// TwinCAT 3 PLC project CNM_ProductionMetrics
// Title: CNM_ProductionMetrics
// Company: ekvip automation GmbH
// Author: tsch
// ProjectVersion: 0.1.1.0
// Description: This library contains classes for measuring and storing production statistics like part counter and cycle time recorder.
// ProgramVersion: 3.1.4026.19
// libraries:
//   CNM_AbstractObject, * (ekvip automation GmbH)
//   CNM_Collections, * (ekvip automation GmbH)
//   CNM_CommandInterfaces, * (ekvip automation GmbH)
//   CNM_ConcreteMessages, * (ekvip automation GmbH)
//   CNM_CycleManager, * (ekvip automation GmbH)
//   CNM_OpModeHandling, * (ekvip automation GmbH)
//   CNM_ProductionMetricInterfaces, * (ekvip automation GmbH)
//   CNM_ReturnTypes, * (ekvip automation GmbH)
//   Tc2_System, * (Beckhoff Automation GmbH)
// project tree:
//   classes/Data/ CycleTimeData.TcPOU, MeasurementData.TcPOU, PartTrackingData.TcPOU
//   classes/Measurements/CycleTimeRecorder/commands/ CycleTimeCaptureCycleCommand.TcPOU, CycleTimeRecorderCommands.TcPOU, CycleTimeStartCycleCommand.TcPOU
//   classes/Measurements/CycleTimeRecorder/ CycleTimeRecorder.TcPOU, CycleTimeRecorderConfiguration.TcPOU
//   classes/Measurements/PartTracking/Commands/ PartTrackingCommands.TcPOU, PartTrackingProcssingStartedCommand.TcPOU, PartTrackingProcssingDoneCommand.TcPOU
//   classes/Measurements/PartTracking/ PartTrackingConfiguration.TcPOU, PartTrackingRecorder.TcPOU
//   classes/Measurements/SimpleMeasurement/commands/ MeasurementAddEntryCommand.TcPOU, MeasurementRecorderCommands.TcPOU
//   classes/Measurements/SimpleMeasurement/ DefaultMeasurementConfiguration.TcPOU, MeasurementRecorder.TcPOU
//   Functions/ GetCurrentLTimeStamp.TcPOU
//   Project Information/ F_GetCompany.TcPOU, F_GetTitle.TcPOU, F_GetVersion.TcPOU
//   / Settings.TcGVL
//   Version/ Global_Version.TcGVL

// ---- Settings.TcGVL
{attribute 'qualified_only'}
VAR_GLOBAL CONSTANT
	(*
	 	The size of the internal queue in the data recorders. 
		when the queue is full, an alarm will be raised and no other 
		dataset will be queued until the list gets emptied 
	*)
	QUEUE_SIZE_FOR_DATA_RECORDS_PER_RECORDER :UDINT := 3;
END_VAR

// ---- Version/Global_Version.TcGVL
{attribute 'TcGenerated'}
{attribute 'no-analysis'}
{attribute 'linkalways'}
// This function has been automatically generated from the project information.
VAR_GLOBAL CONSTANT
	{attribute 'const_non_replaced'}
	stLibVersion_CNM_ProductionMetrics : ST_LibVersion := (iMajor := 0, iMinor := 1, iBuild := 1, iRevision := 0, nFlags := 0, sVersion := '0.1.1.0');
END_VAR

// ---- classes/Data/CycleTimeData.TcPOU
(*

## Short summary

This class serves as a pure data transfer object and can be used to create a new cycle time data set.
An instance of this class can be appended to a production data set list.

.. <legal notes>

legal notes
=================
| SPDX-FileCopyrightText: © 2022 ekvip automation GmbH <info@ekvip.de>
| SPDX-License-Identifier: Apache-2.0
| For details check: Apache-2.0_

.. _Apache-2.0: https://www.apache.org/licenses/LICENSE-2.0

.. </legal notes>

*)
{attribute 'enable_dynamic_creation'}
FUNCTION_BLOCK CycleTimeData EXTENDS CNM_AbstractObject.Object IMPLEMENTS CNM_ProductionMetricInterfaces.ICycleTimeData
VAR
	data :CNM_ProductionMetricInterfaces.CycleTimeDataStruct;
END_VAR

(*

## Short summary

This abstract property returns the class name of the concrete object, 
which is useful for logging/debugging purpose or to check the class name
for ``__DELETE`` in factories (sometimes it's necessary to do more 
than just to free the memory).

.. <legal notes>

legal notes
=================
| SPDX-FileCopyrightText: © 2022 ekvip automation GmbH <info@ekvip.de>
| SPDX-License-Identifier: Apache-2.0
| For details check: Apache-2.0_

.. _Apache-2.0: https://www.apache.org/licenses/LICENSE-2.0

.. </legal notes>

*)
PROPERTY className : CNM_AbstractObject.ClassName
GET
className := 'CycleTimeData';
END_GET
END_PROPERTY

PROPERTY dataset : CNM_ProductionMetricInterfaces.CycleTimeDataStruct
GET
dataset := THIS^.data;
END_GET
END_PROPERTY

(*

## Short summary

The constructor ``FB_init`` is needed to create an unique hash code.
The hash code is a pseudo random number create with a [xorshift](https://en.wikipedia.org/wiki/Xorshift) algorithm.
It can be overwritten on derivations, because it will be called implicit, ``SUPER^.FB_init()`` is not required.
For more information check: [Behavoir with derived function blocks](https://infosys.beckhoff.com/content/1033/tc3_plc_intro/5482088715.html?id=6983869892358031022)

.. <legal notes>

legal notes
=================
| SPDX-FileCopyrightText: © 2022 ekvip automation GmbH <info@ekvip.de>
| SPDX-License-Identifier: Apache-2.0
| For details check: Apache-2.0_

.. _Apache-2.0: https://www.apache.org/licenses/LICENSE-2.0

.. </legal notes>



*)
METHOD FB_init : BOOL
VAR_INPUT
	(* if TRUE, the retain variables are initialized (warm start / cold start)*)
	bInitRetains	: BOOL;
	(* if TRUE, the instance afterwards gets moved into the copy code (online change) *)
	bInCopyCode	: BOOL;
	(* the data set this instance should capsulate *)
	data :CNM_ProductionMetricInterfaces.CycleTimeDataStruct;
END_VAR
THIS^.data := data;
END_METHOD

END_FUNCTION_BLOCK

// ---- classes/Data/MeasurementData.TcPOU
(*
## Short summary

This class serves as a pure data transfer object and can be used to create a new measurement data set.
An instance of this class can be appended to a production data set list.

.. <legal notes>

legal notes
=================
| SPDX-FileCopyrightText: © 2022 ekvip automation GmbH <info@ekvip.de>
| SPDX-License-Identifier: Apache-2.0
| For details check: Apache-2.0_

.. _Apache-2.0: https://www.apache.org/licenses/LICENSE-2.0

.. </legal notes>

*)
{attribute 'enable_dynamic_creation'}
FUNCTION_BLOCK MeasurementData EXTENDS CNM_AbstractObject.Object IMPLEMENTS CNM_ProductionMetricInterfaces.IMeasurementData
VAR
	data : CNM_ProductionMetricInterfaces.MeasurementEntryStruct;
END_VAR

(*

## Short summary

This abstract property returns the class name of the concrete object, 
which is useful for logging/debugging purpose or to check the class name
for ``__DELETE`` in factories (sometimes it's necessary to do more 
than just to free the memory).

.. <legal notes>

legal notes
=================
| SPDX-FileCopyrightText: © 2022 ekvip automation GmbH <info@ekvip.de>
| SPDX-License-Identifier: Apache-2.0
| For details check: Apache-2.0_

.. _Apache-2.0: https://www.apache.org/licenses/LICENSE-2.0

.. </legal notes>

*)
PROPERTY className : CNM_AbstractObject.ClassName
GET
className := 'MeasurementData';
END_GET
END_PROPERTY

(*
## Short summary

This property returns a measurement data set.

.. <legal notes>

legal notes
=================
| SPDX-FileCopyrightText: © 2025 ekvip automation GmbH <info@ekvip.de>
| SPDX-License-Identifier: Apache-2.0
| For details check: Apache-2.0_

.. _Apache-2.0: https://www.apache.org/licenses/LICENSE-2.0

.. </legal notes>

*)
PROPERTY dataset : CNM_ProductionMetricInterfaces.MeasurementEntryStruct
GET
dataset := THIS^.data;
END_GET
END_PROPERTY

(*

## Short summary

The constructor ``FB_init`` is needed to create an unique hash code.
The hash code is a pseudo random number create with a [xorshift](https://en.wikipedia.org/wiki/Xorshift) algorithm.
It can be overwritten on derivations, because it will be called implicit, ``SUPER^.FB_init()`` is not required.
For more information check: [Behavoir with derived function blocks](https://infosys.beckhoff.com/content/1033/tc3_plc_intro/5482088715.html?id=6983869892358031022)

.. <legal notes>

legal notes
=================
| SPDX-FileCopyrightText: © 2022 ekvip automation GmbH <info@ekvip.de>
| SPDX-License-Identifier: Apache-2.0
| For details check: Apache-2.0_

.. _Apache-2.0: https://www.apache.org/licenses/LICENSE-2.0

.. </legal notes>



*)
METHOD FB_init : BOOL
VAR_INPUT
	(* if TRUE, the retain variables are initialized (warm start / cold start)*)
	bInitRetains	: BOOL;
	(* if TRUE, the instance afterwards gets moved into the copy code (online change) *)
	bInCopyCode	: BOOL;
	(* the data set this instance should capsulate *)
	data :CNM_ProductionMetricInterfaces.MeasurementEntryStruct;
END_VAR
THIS^.data := data;
END_METHOD

END_FUNCTION_BLOCK

// ---- classes/Data/PartTrackingData.TcPOU
(*

## Short summary

This class serves as a pure data transfer object and can be used to create a new part counter data set.
An instance of this class can be appended to a production data set list.

.. <legal notes>

legal notes
=================
| SPDX-FileCopyrightText: © 2022 ekvip automation GmbH <info@ekvip.de>
| SPDX-License-Identifier: Apache-2.0
| For details check: Apache-2.0_

.. _Apache-2.0: https://www.apache.org/licenses/LICENSE-2.0

.. </legal notes>

*)
{attribute 'enable_dynamic_creation'}
FUNCTION_BLOCK PartTrackingData EXTENDS CNM_AbstractObject.Object IMPLEMENTS CNM_ProductionMetricInterfaces.IPartTrackingData
VAR
	data :CNM_ProductionMetricInterfaces.PartDataTrackingStruct;
END_VAR

(*

## Short summary

This abstract property returns the class name of the concrete object, 
which is useful for logging/debugging purpose or to check the class name
for ``__DELETE`` in factories (sometimes it's necessary to do more 
than just to free the memory).

.. <legal notes>

legal notes
=================
| SPDX-FileCopyrightText: © 2022 ekvip automation GmbH <info@ekvip.de>
| SPDX-License-Identifier: Apache-2.0
| For details check: Apache-2.0_

.. _Apache-2.0: https://www.apache.org/licenses/LICENSE-2.0

.. </legal notes>

*)
PROPERTY className : CNM_AbstractObject.ClassName
GET
className := 'PartCounterData';
END_GET
END_PROPERTY

PROPERTY dataset : CNM_ProductionMetricInterfaces.PartDataTrackingStruct
GET
dataset := THIS^.data;
END_GET
END_PROPERTY

(*

## Short summary

The constructor ``FB_init`` is needed to create an unique hash code.
The hash code is a pseudo random number create with a [xorshift](https://en.wikipedia.org/wiki/Xorshift) algorithm.
It can be overwritten on derivations, because it will be called implicit, ``SUPER^.FB_init()`` is not required.
For more information check: [Behavoir with derived function blocks](https://infosys.beckhoff.com/content/1033/tc3_plc_intro/5482088715.html?id=6983869892358031022)

.. <legal notes>

legal notes
=================
| SPDX-FileCopyrightText: © 2022 ekvip automation GmbH <info@ekvip.de>
| SPDX-License-Identifier: Apache-2.0
| For details check: Apache-2.0_

.. _Apache-2.0: https://www.apache.org/licenses/LICENSE-2.0

.. </legal notes>



*)
METHOD FB_init : BOOL
VAR_INPUT
	(* if TRUE, the retain variables are initialized (warm start / cold start)*)
	bInitRetains	: BOOL;
	(* if TRUE, the instance afterwards gets moved into the copy code (online change) *)
	bInCopyCode	: BOOL;
	(* the data set this instance should capsulate *)
	data :CNM_ProductionMetricInterfaces.PartDataTrackingStruct;
END_VAR
THIS^.data := data;
END_METHOD

END_FUNCTION_BLOCK

// ---- classes/Measurements/CycleTimeRecorder/commands/CycleTimeCaptureCycleCommand.TcPOU
(*
## Short summary

This command can be used to set the cycle start timestamp manually.

**Attention:** If only the captureCurrentCycle method is called, the start timestamp will be set automatically when the previous cycle is done.

.. <legal notes>

legal notes
=================
| SPDX-FileCopyrightText: © 2025 ekvip automation GmbH <info@ekvip.de>
| SPDX-License-Identifier: Apache-2.0
| For details check: Apache-2.0_

.. _Apache-2.0: https://www.apache.org/licenses/LICENSE-2.0

.. </legal notes>

*)
FUNCTION_BLOCK CycleTimeCaptureCycleCommand EXTENDS CNM_AbstractObject.Object IMPLEMENTS CNM_CommandInterfaces.ISingleAttempt
VAR
	recorder :CNM_ProductionMetricInterfaces.ICycleTimeRecorder;
	additionalMessage :Tc2_System.T_MaxString := '';
END_VAR

(*

## Short summary

This abstract property returns the class name of the concrete object, 
which is useful for logging/debugging purpose or to check the class name
for ``__DELETE`` in factories (sometimes it's necessary to do more 
than just to free the memory).

.. <legal notes>

legal notes
=================
| SPDX-FileCopyrightText: © 2022 ekvip automation GmbH <info@ekvip.de>
| SPDX-License-Identifier: Apache-2.0
| For details check: Apache-2.0_

.. _Apache-2.0: https://www.apache.org/licenses/LICENSE-2.0

.. </legal notes>

*)
PROPERTY className : CNM_AbstractObject.ClassName
GET
className :=  'CNM_ProductionMetrics.CycleTimeCaptureCycleCommand';
END_GET
END_PROPERTY

(*

## Short summary

Invokes the action associated with this interface.

.. <legal notes>

legal notes
=================
| SPDX-FileCopyrightText: © 2024 ekvip automation GmbH <info@ekvip.de>
| SPDX-License-Identifier: Apache-2.0
| For details check: Apache-2.0_

.. _Apache-2.0: https://www.apache.org/licenses/LICENSE-2.0

.. </legal notes>



*)
METHOD invoke : CNM_ReturnTypes.SingleExecutionResult
IF THIS^.isObjectValid(THIS^.recorder) THEN
	invoke := THIS^.recorder.captureCurrentCycle(additionalMessage := THIS^.additionalMessage);
ELSE
	invoke := CNM_ReturnTypes.SingleExecutionResult.ABORTED;
END_IF
END_METHOD

METHOD INTERNAL setParameters
VAR_INPUT
	(* can be used to provide additional informations for the record, e.g. multiple measurements neccesray or test part *)
	additionalMessage	:Tc2_System.T_MaxString := '';
END_VAR
THIS^.additionalMessage := additionalMessage;
END_METHOD

(*
## Short summary

This methods sets the cycletime recorder interface on which the command is executed.

.. <legal notes>

legal notes
=================
| SPDX-FileCopyrightText: © 2025 ekvip automation GmbH <info@ekvip.de>
| SPDX-License-Identifier: Apache-2.0
| For details check: Apache-2.0_

.. _Apache-2.0: https://www.apache.org/licenses/LICENSE-2.0

.. </legal notes>

*)

METHOD INTERNAL setRecorder
VAR_INPUT
	recorder :CNM_ProductionMetricInterfaces.ICycleTimeRecorder;
END_VAR
IF THIS^.isObjectValid(recorder) THEN
	THIS^.recorder := recorder;
END_IF
END_METHOD

END_FUNCTION_BLOCK

// ---- classes/Measurements/CycleTimeRecorder/commands/CycleTimeRecorderCommands.TcPOU
(* 
## Short summary

This class is a collection of cycle time recorder commands that provides a fluent interface for single attempt commands, which can be evaluated by a cycle manager instance.
### Example 
```
	cycleManager.leave(
		cycleTimeRecorder.commands.captureCurrentCycle(
			additionalMessage := 'just an example'
		)
	);  
	```

.. <legal notes>

legal notes
=================
| SPDX-FileCopyrightText: © 2025 ekvip automation GmbH <info@ekvip.de>
| SPDX-License-Identifier: Apache-2.0
| For details check: Apache-2.0_

.. _Apache-2.0: https://www.apache.org/licenses/LICENSE-2.0

.. </legal notes>
	
*)

FUNCTION_BLOCK CycleTimeRecorderCommands EXTENDS CNM_AbstractObject.Object IMPLEMENTS CNM_ProductionMetricInterfaces.ICycleTimeRecorderCommands
VAR
	captureCommand :CycleTimeCaptureCycleCommand;
	startCycleCommand :CycleTimeStartCycleCommand;
END_VAR

(*

## Short summary

This command creates a new cycle time roecord for the currently produced part by calculating the the passed time since the last call of this method.
If a new mode is started the last timestamp will be set to the moment when the mode was started.


.. <legal notes>

legal notes
=================
| SPDX-FileCopyrightText: © 2025 ekvip automation GmbH <info@ekvip.de>
| SPDX-License-Identifier: Apache-2.0
| For details check: Apache-2.0_

.. _Apache-2.0: https://www.apache.org/licenses/LICENSE-2.0

.. </legal notes>

*)
METHOD captureCurrentCycle : CNM_CommandInterfaces.ISingleAttempt
VAR_INPUT
	(* can be used to provide additional informations for the record, e.g. multiple measurements neccesray or test part *)
	additionalMessage	: Tc2_System.T_MaxString := '';
END_VAR
THIS^.captureCommand.setParameters(additionalMessage);
captureCurrentCycle := THIS^.captureCommand;
END_METHOD

(*

## Short summary

This abstract property returns the class name of the concrete object, 
which is useful for logging/debugging purpose or to check the class name
for ``__DELETE`` in factories (sometimes it's necessary to do more 
than just to free the memory).

.. <legal notes>

legal notes
=================
| SPDX-FileCopyrightText: © 2022 ekvip automation GmbH <info@ekvip.de>
| SPDX-License-Identifier: Apache-2.0
| For details check: Apache-2.0_

.. _Apache-2.0: https://www.apache.org/licenses/LICENSE-2.0

.. </legal notes>

*)

PROPERTY className : CNM_AbstractObject.ClassName
GET
 className := 'CNM_ProductionMetrics.CycleTimeRecorderCommands';
END_GET
END_PROPERTY

METHOD INTERNAL setRecorder : BOOL
VAR_INPUT
	recorder :CNM_ProductionMetricInterfaces.ICycleTimeRecorder;
END_VAR
IF THIS^.isObjectValid(recorder) THEN
	THIS^.captureCommand.setRecorder(recorder);
	THIS^.startCycleCommand.setRecorder(recorder);
END_IF
END_METHOD

(*
## Short summary

This command can be used to set the cycle start timestamp manually.

**Attention:** If only the captureCurrentCycle method is called, the start timestamp will be set automatically when the previous cycle is done.

.. <legal notes>

legal notes
=================
| SPDX-FileCopyrightText: © 2025 ekvip automation GmbH <info@ekvip.de>
| SPDX-License-Identifier: Apache-2.0
| For details check: Apache-2.0_

.. _Apache-2.0: https://www.apache.org/licenses/LICENSE-2.0

.. </legal notes>

*)
METHOD startCycle : CNM_CommandInterfaces.ISingleAttempt
startCycle := THIS^.startCycleCommand;
END_METHOD

END_FUNCTION_BLOCK

// ---- classes/Measurements/CycleTimeRecorder/commands/CycleTimeStartCycleCommand.TcPOU
(*
## Short summary

This command can be used to set the cycle start timestamp manually.

**Attention:** If only the captureCurrentCycle method is called, the start timestamp will be set automatically when the previous cycle is done.

.. <legal notes>

legal notes
=================
| SPDX-FileCopyrightText: © 2025 ekvip automation GmbH <info@ekvip.de>
| SPDX-License-Identifier: Apache-2.0
| For details check: Apache-2.0_

.. _Apache-2.0: https://www.apache.org/licenses/LICENSE-2.0

.. </legal notes>

*)
FUNCTION_BLOCK CycleTimeStartCycleCommand EXTENDS CNM_AbstractObject.Object IMPLEMENTS CNM_CommandInterfaces.ISingleAttempt
VAR
	recorder :CNM_ProductionMetricInterfaces.ICycleTimeRecorder;
END_VAR

(*

## Short summary

This abstract property returns the class name of the concrete object, 
which is useful for logging/debugging purpose or to check the class name
for ``__DELETE`` in factories (sometimes it's necessary to do more 
than just to free the memory).

.. <legal notes>

legal notes
=================
| SPDX-FileCopyrightText: © 2022 ekvip automation GmbH <info@ekvip.de>
| SPDX-License-Identifier: Apache-2.0
| For details check: Apache-2.0_

.. _Apache-2.0: https://www.apache.org/licenses/LICENSE-2.0

.. </legal notes>

*)
PROPERTY className : CNM_AbstractObject.ClassName
GET
className := 'CNM_ProductionMetrics.CycleTimeStartCycleCommand';
END_GET
END_PROPERTY

(*

## Short summary

Invokes the action associated with this interface.

.. <legal notes>

legal notes
=================
| SPDX-FileCopyrightText: © 2024 ekvip automation GmbH <info@ekvip.de>
| SPDX-License-Identifier: Apache-2.0
| For details check: Apache-2.0_

.. _Apache-2.0: https://www.apache.org/licenses/LICENSE-2.0

.. </legal notes>



*)
METHOD invoke : CNM_ReturnTypes.SingleExecutionResult
IF THIS^.isObjectValid(THIS^.recorder) THEN
	invoke := THIS^.recorder.startCycle();
ELSE
	invoke := CNM_ReturnTypes.SingleExecutionResult.ABORTED;
END_IF
END_METHOD

(*
## Short summary

This methods sets the cycletime recorder interface on which the command is executed.

.. <legal notes>

legal notes
=================
| SPDX-FileCopyrightText: © 2025 ekvip automation GmbH <info@ekvip.de>
| SPDX-License-Identifier: Apache-2.0
| For details check: Apache-2.0_

.. _Apache-2.0: https://www.apache.org/licenses/LICENSE-2.0

.. </legal notes>

*)

METHOD setRecorder
VAR_INPUT
	recorder :CNM_ProductionMetricInterfaces.ICycleTimeRecorder;
END_VAR
IF THIS^.isObjectValid(recorder) THEN
	THIS^.recorder := recorder;
END_IF
END_METHOD

END_FUNCTION_BLOCK

// ---- classes/Measurements/CycleTimeRecorder/CycleTimeRecorder.TcPOU
(*
## Short summary

This class provides the functionalities to measure timespans for processes and commands.
It can measure processing times (start time -> stop time) and cycle times (last stop time -> stop time).

.. <legal notes>

legal notes
=================
| SPDX-FileCopyrightText: © 2025 ekvip automation GmbH <info@ekvip.de>
| SPDX-License-Identifier: Apache-2.0
| For details check: Apache-2.0_

.. _Apache-2.0: https://www.apache.org/licenses/LICENSE-2.0

.. </legal notes>

*)

FUNCTION_BLOCK CycleTimeRecorder EXTENDS CNM_OpModeHandler.AbstractCyclicNode IMPLEMENTS CNM_ProductionMetricInterfaces.ICycleTimeRecorder
VAR
	(* current data *)
	currentCycleTimeData :CNM_ProductionMetricInterfaces.CycleTimeDataStruct;
	(* queue for the measurements *)
	dataSetList :CNM_Collections.LinkedList;
	(* the variable that is used as data slot to provide data for the database *)
	{ attribute 'TcHmiSymbol.ShowRecursively' }
	cycleTimeRecord :CNM_ProductionMetricInterfaces.CycleTimeDataStruct;
	(* mailbox flag for the database that we have a new entry, should be reset by the server when data was read *)
	{ attribute 'TcHmiSymbol.Show' }
	newDataAvailable :BOOL := FALSE;
	(* command delegates *)
	cycleTimeCommands :CycleTimeRecorderCommands;
	(* error for failed queryInterface *)
	interfaceQueryFailedAlarm :CNM_ConcreteMessages.TcError(
		event := Global.TC_EVENTS.MemoryErrors.CycleTimeRecorderQueryInterfacFailed , 
		injectedService := THIS^.messageService
	); 
	(* error for maximum queue size *)
	maxQueueSizeAlarm :CNM_ConcreteMessages.TcError(event := Global.TC_EVENTS.MemoryErrors.CycleTimeMaxQueueSize, injectedService := THIS^.messageService);
END_VAR

(*

## Short summary

This method creates a new cycle time roecord for the currently produced part by calculating the the passed time since the last call of this method.
If a new mode is started the last timestamp will be set to the moment when the mode was started.


.. <legal notes>

legal notes
=================
| SPDX-FileCopyrightText: © 2025 ekvip automation GmbH <info@ekvip.de>
| SPDX-License-Identifier: Apache-2.0
| For details check: Apache-2.0_

.. _Apache-2.0: https://www.apache.org/licenses/LICENSE-2.0

.. </legal notes>

*)
METHOD captureCurrentCycle : CNM_ProductionMetricInterfaces.CNM_ReturnTypes.SingleExecutionResult
VAR_INPUT
	(* can be used to provide additional informations for the record, e.g. multiple measurements neccesray or test part *)
	additionalMessage	: Tc2_System.T_MaxString := '';
END_VAR
VAR
	dto :POINTER TO CycleTimeData;
	(* data backup to restore timestamps *)
	backupEndTimestamp :LDT;
END_VAR
captureCurrentCycle := CNM_ReturnTypes.SingleExecutionResult.ABORTED;
// check if we can queue the dataset - throw error if the max queuesize is reached
IF ( THIS^.dataSetList.size >= THIS^.maxQueueSize ) THEN
	THIS^.maxQueueSizeAlarm.throw();
	RETURN;
END_IF

backupEndTimestamp  := THIS^.currentCycleTimeData.endTimestamp;
THIS^.currentCycleTimeData.cycleTime := 
	SEL(
		TO_UDINT(THIS^.currentCycleTimeData.endTimestamp) > 0, 
		TO_LTIME(0), 
		TO_LTIME(GetCurrentLTimeStamp() - THIS^.currentCycleTimeData.endTimestamp ));
THIS^.currentCycleTimeData.endTimestamp := GetCurrentLTimeStamp();
THIS^.currentCycleTimeData.processingTime := 
	SEL(
		TO_UDINT(THIS^.currentCycleTimeData.startTimestamp) > 0, 
		TO_LTIME(0), 
		TO_LTIME(THIS^.currentCycleTimeData.endTimestamp - THIS^.currentCycleTimeData.startTimestamp));
THIS^.currentCycleTimeData.process := THIS^.configuration.process;
THIS^.currentCycleTimeData.productType := THIS^.configuration.productType;
THIS^.currentCycleTimeData.targetCycletime := THIS^.configuration.targetCycleTime;
THIS^.currentCycleTimeData.additionalMessage := additionalMessage;
dto := __NEW(CycleTimeData(data := THIS^.currentCycleTimeData));
IF (dto <> 0) THEN
	captureCurrentCycle := THIS^.dataSetList.append(dto^);
ELSE
	// restore data for retry
	THIS^.currentCycleTimeData.endTimestamp := backupEndTimestamp;
END_IF
END_METHOD

(*

## Short summary

This abstract property returns the class name of the concrete object, 
which is useful for logging/debugging purpose or to check the class name
for ``__DELETE`` in factories (sometimes it's necessary to do more 
than just to free the memory).

.. <legal notes>

legal notes
=================
| SPDX-FileCopyrightText: © 2022 ekvip automation GmbH <info@ekvip.de>
| SPDX-License-Identifier: Apache-2.0
| For details check: Apache-2.0_

.. _Apache-2.0: https://www.apache.org/licenses/LICENSE-2.0

.. </legal notes>

*)
PROPERTY className : CNM_AbstractObject.ClassName
GET
className := 'CycleTimeRecorder';
END_GET
END_PROPERTY

(* 
## Short summary

This is a fluent interface that provides single attempt commands, which can be evaluated by a cycle manager instance.
### Example 
```
	cycleManager.leave(
		cycleTimeRecorder.commands.captureCurrentCycle(
			additionalMessage := 'just an example'
		)
	);  
	```

.. <legal notes>

legal notes
=================
| SPDX-FileCopyrightText: © 2025 ekvip automation GmbH <info@ekvip.de>
| SPDX-License-Identifier: Apache-2.0
| For details check: Apache-2.0_

.. _Apache-2.0: https://www.apache.org/licenses/LICENSE-2.0

.. </legal notes>
	
*)

PROPERTY commands : CNM_ProductionMetricInterfaces.ICycleTimeRecorderCommands
GET
commands := THIS^.cycleTimeCommands;
END_GET
END_PROPERTY

(*
## Short summary

This property returns an fluent interface for the cycle time recorder configuration.
The following things should be configured after a type / product / batch change was performed:
 -product type: either the name of the overall product or the individual feed parts to be processed
 -targetCycleTime: the target cycle time for this process and product type
 
The process name can be set once during the initialization of the PLC as it usually doesn't change.

.. <legal notes>

legal notes
=================
| SPDX-FileCopyrightText: © 2025 ekvip automation GmbH <info@ekvip.de>
| SPDX-License-Identifier: Apache-2.0
| For details check: Apache-2.0_

.. _Apache-2.0: https://www.apache.org/licenses/LICENSE-2.0

.. </legal notes>

*)
PROPERTY configuration : CNM_ProductionMetricInterfaces.ICycleTimeConfiguration
GET
VAR_INST
	config :CycleTimeRecorderConfiguration;
END_VAR
configuration := config;
END_GET
END_PROPERTY

(* 
## Short summary

This method disables a node (E.g. axes should be disabled). It can take mutliple cycles. It has to be implemented for every node/device.
The execute input needs a rising edge to execute the method.
If there is nothing to disable, just return a 'SUCCESS' state.

This method is called automatically by the operation mode handler.

.. <legal notes>

legal notes
=================
| SPDX-FileCopyrightText: © 2024 ekvip automation GmbH <info@ekvip.de>
| SPDX-License-Identifier: Apache-2.0
| For details check: Apache-2.0_

.. _Apache-2.0: https://www.apache.org/licenses/LICENSE-2.0

.. </legal notes>

*)
METHOD disable : CNM_ReturnTypes.SingleExecutionState
VAR_INPUT
	execute	: BOOL;
END_VAR
// nothing to disable
disable := CNM_ReturnTypes.SingleExecutionState.SUCCESS;
END_METHOD

(* 
## Short summary

This method enables a node. It can take mutliple cycles. It has to be implemented for every node/device.
The intention is to enable devices here, e.g. axes, laser, dispenser etc.
The execute input needs a rising edge to execute the method.
If there is nothing to enable, just return a 'SUCCESS' state.

This method is called automatically by the operation mode handler.

.. <legal notes>

legal notes
=================
| SPDX-FileCopyrightText: © 2024 ekvip automation GmbH <info@ekvip.de>
| SPDX-License-Identifier: Apache-2.0
| For details check: Apache-2.0_

.. _Apache-2.0: https://www.apache.org/licenses/LICENSE-2.0

.. </legal notes>

*)
METHOD enable : CNM_ReturnTypes.SingleExecutionState
VAR_INPUT
	execute	: BOOL;
END_VAR
// nothing to enable
enable := CNM_ReturnTypes.SingleExecutionState.SUCCESS;
END_METHOD

(*

## Short summary

The constructor ``FB_init`` is needed to create an unique hash code.
The hash code is a pseudo random number create with a [xorshift](https://en.wikipedia.org/wiki/Xorshift) algorithm.
It can be overwritten on derivations, because it will be called implicit, ``SUPER^.FB_init()`` is not required.
For more information check: [Behavoir with derived function blocks](https://infosys.beckhoff.com/content/1033/tc3_plc_intro/5482088715.html?id=6983869892358031022)

.. <legal notes>

legal notes
=================
| SPDX-FileCopyrightText: © 2022 ekvip automation GmbH <info@ekvip.de>
| SPDX-License-Identifier: Apache-2.0
| For details check: Apache-2.0_

.. _Apache-2.0: https://www.apache.org/licenses/LICENSE-2.0

.. </legal notes>



*)
METHOD FB_init : BOOL
VAR_INPUT
	(* if TRUE, the retain variables are initialized (warm start / cold start)*)
	bInitRetains	: BOOL;
	(* if TRUE, the instance afterwards gets moved into the copy code (online change) *)
	bInCopyCode	:BOOL;
	(* the node were this node should be appended to *)
	parentNode :CNM_OpModeHandler.INodeInitialization;
END_VAR
THIS^.hmiInfo.template := 'TimeTrackingRecorder';
THIS^.isInHome := TRUE;
END_METHOD

(* 
## Short summary

This method contains instructions and sequences for the init mode. 
This mode is intended for initializing a machine, e.g. loading product type data from recipes, establish a connection to global production systems (MES).
If the node should do nothing, return a 'SUCCESS'.
It should run until all initializations are done or the mode is stopped immedtiately or a stop request is raised (THIS^.modeControl.stopRequest). 
This method is called automatically by the operation mode handler.

**Attention:** If this method returns the state 'ERROR', the operation mode handler automatically disables the whole machine! 

.. <legal notes>

legal notes
=================
| SPDX-FileCopyrightText: © 2024 ekvip automation GmbH <info@ekvip.de>
| SPDX-License-Identifier: Apache-2.0
| For details check: Apache-2.0_

.. _Apache-2.0: https://www.apache.org/licenses/LICENSE-2.0

.. </legal notes>

*)
METHOD initialize : CNM_ReturnTypes.SingleExecutionState
VAR_INPUT
	execute	: BOOL;
END_VAR
THIS^.cycleTimeCommands.setRecorder(THIS^);
initialize := CNM_ReturnTypes.SingleExecutionState.SUCCESS;
END_METHOD

(*
## Short summary

This property getter returns the maximum queue size for the data recorder. 
If the dataset list has reached this size, no other dataset will be stored and an alarm will be raised.
For this class the maximum queue size can be configured as library parameter ''QUEUE_SIZE_FOR_DATA_RECORDS_PER_RECORDER''.
Overwrite this property for extended classes as the default implementation accesses the Parameter List of the CNM_ProductionMetrics library! 

.. <legal notes>

legal notes
=================
| SPDX-FileCopyrightText: © 2022 ekvip automation GmbH <info@ekvip.de>
| SPDX-License-Identifier: Apache-2.0
| For details check: Apache-2.0_

.. _Apache-2.0: https://www.apache.org/licenses/LICENSE-2.0

.. </legal notes>

*)

PROPERTY PROTECTED maxQueueSize : UDINT
GET
maxQueueSize := Settings.QUEUE_SIZE_FOR_DATA_RECORDS_PER_RECORDER;
END_GET
END_PROPERTY

(* 
## Short summary

This method will be called in every cycle for a node. It can be used to implement hardware drivers/measurements/monitoring.
The returned state defines the overall state of the node. It should return BUSY when the node executes a command, otherwise SUCCESS( or IDLE if there is nothing to do). 
(Simple monitoring is not a command an should return SUCCESS).  


**Attention:** the returned SingleExecutionState will be evaluated cyclically wihtin the node tree. 
In case a node returns an ERROR state, the whole machine will be disabled. 
Return ERROR only for fatal or critical errors and handle other errors within the node.
 

.. <legal notes>

legal notes
=================
| SPDX-FileCopyrightText: © 2025 ekvip automation GmbH <info@ekvip.de>
| SPDX-License-Identifier: Apache-2.0
| For details check: Apache-2.0_

.. _Apache-2.0: https://www.apache.org/licenses/LICENSE-2.0

.. </legal notes>
	
*)
METHOD run : CNM_ReturnTypes.SingleExecutionState
VAR_INST
	cycleManager :CNM_CycleManager.SimpleCycleManager;
END_VAR
VAR CONSTANT
	WAIT_FOR_DATA :DINT := 10;
	SET_DATA :DINT := 11;
	DATA_ERROR :DINT := 12;
	WAIT_DATA_RECEIVED :DINT := 13;
END_VAR
VAR
	data :CNM_ProductionMetricInterfaces.ICycleTimeData;
END_VAR
cycleManager(execute := TRUE);

CASE cycleManager.step.current OF
CNM_ReturnTypes.DefaultSteps.STEP.INIT:
	run := CNM_ReturnTypes.SingleExecutionState.SUCCESS;
	cycleManager.proceedWith(WAIT_FOR_DATA);
WAIT_FOR_DATA:
	run := CNM_ReturnTypes.SingleExecutionState.SUCCESS;
	IF (THIS^.dataSetList.size > 0) THEN
		run := CNM_ReturnTypes.SingleExecutionState.BUSY;
		cycleManager.proceedWith(SET_DATA); 
	END_IF
SET_DATA:
	run := CNM_ReturnTypes.SingleExecutionState.BUSY;
	IF (__QUERYINTERFACE(THIS^.dataSetList.dequeue(), data)) THEN
		(* fill dataslot *)
		THIS^.cycleTimeRecord := data.dataset;
		(* delete DTO *)
		data.destruct();
		(* set mailbox flag *)
		THIS^.newDataAvailable := TRUE;
		cycleManager.proceedWith(WAIT_DATA_RECEIVED);
	ELSE
		cycleManager.proceedWith(DATA_ERROR);
	END_IF
DATA_ERROR:
	cycleManager.step.next := SET_DATA;
	cycleManager.handle(THIS^.interfaceQueryFailedAlarm);
WAIT_DATA_RECEIVED:
	run := CNM_ReturnTypes.SingleExecutionState.BUSY;
	IF (NOT THIS^.newDataAvailable) THEN
		// clear data slot
		Tc2_System.MEMSET(destAddr := ADR(THIS^.cycleTimeRecord), 0, SIZEOF(THIS^.cycleTimeRecord));
		run := CNM_ReturnTypes.SingleExecutionState.SUCCESS;
		cycleManager.proceedWith(WAIT_FOR_DATA);
	END_IF
END_CASE
END_METHOD

(*
## Short summary

This method can be used to set the cycle start timestamp manually.

**Attention:** If only the captureCurrentCycle method is called, the start timestamp will be set automatically when the previous cycle is done.

.. <legal notes>

legal notes
=================
| SPDX-FileCopyrightText: © 2025 ekvip automation GmbH <info@ekvip.de>
| SPDX-License-Identifier: Apache-2.0
| For details check: Apache-2.0_

.. _Apache-2.0: https://www.apache.org/licenses/LICENSE-2.0

.. </legal notes>

*)
METHOD startCycle :CNM_ReturnTypes.SingleExecutionResult;
THIS^.currentCycleTimeData.startTimestamp := GetCurrentLTimeStamp();
startCycle := CNM_ReturnTypes.SingleExecutionResult.SUCCESS;
END_METHOD

(* 
## Short summary

This method executes stops all movements of a node. It has to be overwritten for every node. 
E.g. axes should perform a quickstop, cylinders should be turned off, etc.
If the node should do nothing, return a 'SUCCESS'.
It should stop axes/cylinders/process (e.g. laser welding, dispensing) endless until the manual mode is stopped via stop request or immediate stop.
This method is called automatically by the operation mode handler before disabling the machine or if the operator selects an immediate stop.

**Attention:** If this method returns the state 'ERROR', the operation mode handler automatically disables the whole machine! 

.. <legal notes>

legal notes
=================
| SPDX-FileCopyrightText: © 2024 ekvip automation GmbH <info@ekvip.de>
| SPDX-License-Identifier: Apache-2.0
| For details check: Apache-2.0_

.. _Apache-2.0: https://www.apache.org/licenses/LICENSE-2.0

.. </legal notes>

*)
METHOD stopImmediate : CNM_ReturnTypes.SingleExecutionState
VAR_INPUT
	execute	: BOOL;
END_VAR
// nothing to stop
stopImmediate := CNM_ReturnTypes.SingleExecutionState.SUCCESS;
END_METHOD

END_FUNCTION_BLOCK

// ---- Functions/GetCurrentLTimeStamp.TcPOU
(* 
The issue when getting timestamps: two different base times

The function F_GetSystemTime returns the current time in 100 nanosecond steps as ULINT since 1.1.1601 (Windows base time)
The LDATE_AND_TIME type starts on the UNIX base time - 1.1.1970. 
  
To get the correct time in the end, we have to subtract the difference of 369 years or 11644473600 seconds.
  *)

FUNCTION GetCurrentLTimeStamp : LDATE_AND_TIME
VAR CONSTANT
	(* 369 years in seconds, the difference between UNIX starttime (1970) and windows starttime (1601) *)
	CORRECTION	: ULINT := 11644473600;
END_VAR

(* current time in 100 nanoseconds since 1970 * 100  -  the correction in nanoseconds *)
GetCurrentLTimeStamp := TO_LDT(F_GetSystemTime()*100 - CORRECTION*TO_ULINT(1E9));

END_FUNCTION

// ---- classes/Measurements/CycleTimeRecorder/CycleTimeRecorderConfiguration.TcPOU
(* 
## Short summary

This class is a data transfer object for configurable cycle time recorder attributes. 
It is intended to be uses within a fluid configuration interface. 

.. <legal notes>

legal notes
=================
| SPDX-FileCopyrightText: © 2025 ekvip automation GmbH <info@ekvip.de>
| SPDX-License-Identifier: Apache-2.0
| For details check: Apache-2.0_

.. _Apache-2.0: https://www.apache.org/licenses/LICENSE-2.0

.. </legal notes>

*)

FUNCTION_BLOCK CycleTimeRecorderConfiguration EXTENDS DefaultMeasurementConfiguration IMPLEMENTS CNM_ProductionMetricInterfaces.ICycleTimeConfiguration
VAR
	configuredTargetCycleTime :LTIME;
END_VAR

(*

## Short summary

This abstract property returns the class name of the concrete object, 
which is useful for logging/debugging purpose or to check the class name
for ``__DELETE`` in factories (sometimes it's necessary to do more 
than just to free the memory).

.. <legal notes>

legal notes
=================
| SPDX-FileCopyrightText: © 2022 ekvip automation GmbH <info@ekvip.de>
| SPDX-License-Identifier: Apache-2.0
| For details check: Apache-2.0_

.. _Apache-2.0: https://www.apache.org/licenses/LICENSE-2.0

.. </legal notes>

*)
PROPERTY className : CNM_AbstractObject.ClassName
GET
className := 'CycleTimeRecorderConfiguration';
END_GET
END_PROPERTY

(* 
## Short summary

This property can be used to set and read the current target cycle time for a product cycle of a single part.
The target cycle time will be written into every measurement entry and is used to mark cycle time exceedances.

.. <legal notes>

legal notes
=================
| SPDX-FileCopyrightText: © 2025 ekvip automation GmbH <info@ekvip.de>
| SPDX-License-Identifier: Apache-2.0
| For details check: Apache-2.0_

.. _Apache-2.0: https://www.apache.org/licenses/LICENSE-2.0

.. </legal notes>

*)
PROPERTY targetCycleTime : LTIME
GET
targetCycleTime := THIS^.configuredTargetCycleTime;
END_GET
SET
THIS^.configuredTargetCycleTime := targetCycleTime;
END_SET
END_PROPERTY

END_FUNCTION_BLOCK

// ---- classes/Measurements/SimpleMeasurement/DefaultMeasurementConfiguration.TcPOU
(* 
## Short summary

This class is a data transfer object that contains the default configuration properties for production measurement configurations.

.. <legal notes>

legal notes
=================
| SPDX-FileCopyrightText: © 2025 ekvip automation GmbH <info@ekvip.de>
| SPDX-License-Identifier: Apache-2.0
| For details check: Apache-2.0_

.. _Apache-2.0: https://www.apache.org/licenses/LICENSE-2.0

.. </legal notes>

*)

FUNCTION_BLOCK DefaultMeasurementConfiguration EXTENDS CNM_AbstractObject.Object IMPLEMENTS CNM_ProductionMetricInterfaces.IProductionMetricsConfiguration
VAR
	configuredProcess :Tc2_System.T_MaxString;
	configuredProductType :Tc2_System.T_MaxString;
END_VAR

(*

## Short summary

This abstract property returns the class name of the concrete object, 
which is useful for debugging purpose or to check the class name for 
``__DELETE`` in factories (sometimes it's necessary to do more 
than just to free the memory).

**Attention:**: 
	For derivations: **It is necessary that this property is overridden by the concrete class**

.. <legal notes>

legal notes
=================
| SPDX-FileCopyrightText: © 2022 ekvip automation GmbH <info@ekvip.de>
| SPDX-License-Identifier: Apache-2.0
| For details check: Apache-2.0_

.. _Apache-2.0: https://www.apache.org/licenses/LICENSE-2.0

.. </legal notes>

*)
PROPERTY className : CNM_AbstractObject.ClassName
GET
className := 'AbstractMeasurementConfiguration';
END_GET
END_PROPERTY

(* 
## Short summary

This property can be used to set and read the process number or name as string.

.. <legal notes>

legal notes
=================
| SPDX-FileCopyrightText: © 2025 ekvip automation GmbH <info@ekvip.de>
| SPDX-License-Identifier: Apache-2.0
| For details check: Apache-2.0_

.. _Apache-2.0: https://www.apache.org/licenses/LICENSE-2.0

.. </legal notes>

*)
PROPERTY FINAL process : Tc2_System.T_MaxString
GET
process := THIS^.configuredProcess;
END_GET
SET
THIS^.configuredProcess := process;
END_SET
END_PROPERTY

(* 
## Short summary

This property can be used to set and read the current product type (TTNR/PTN) as string.
The type will be written into every measurement entry.

.. <legal notes>

legal notes
=================
| SPDX-FileCopyrightText: © 2025 ekvip automation GmbH <info@ekvip.de>
| SPDX-License-Identifier: Apache-2.0
| For details check: Apache-2.0_

.. _Apache-2.0: https://www.apache.org/licenses/LICENSE-2.0

.. </legal notes>

*)
PROPERTY FINAL productType : Tc2_System.T_MaxString
GET
productType := THIS^.configuredProductType;
END_GET
SET
THIS^.configuredProductType := productType;
END_SET
END_PROPERTY

END_FUNCTION_BLOCK

// ---- classes/Measurements/PartTracking/Commands/PartTrackingCommands.TcPOU
(* 
## Short summary

This class is a fluent interface that provides single attempt commands, which can be evaluated by a cycle manager instance.
### Example 
```
	
	// execute command when leaving a step 
	cycleManager.leave(
		partTracker.commands.partProcessingDone(
			partIdentifier := 'Part123',
			nokReason := 0,
			additionalMessage := 'SPC Part'
		)
	);  
```
.. <legal notes>

legal notes
=================
| SPDX-FileCopyrightText: © 2025 ekvip automation GmbH <info@ekvip.de>
| SPDX-License-Identifier: Apache-2.0
| For details check: Apache-2.0_

.. _Apache-2.0: https://www.apache.org/licenses/LICENSE-2.0

.. </legal notes>
	
*)

FUNCTION_BLOCK PartTrackingCommands EXTENDS CNM_AbstractObject.Object IMPLEMENTS CNM_ProductionMetricInterfaces.IPartTrackingRecorderCommands
VAR
	startProcessing :PartTrackingProcssingStartedCommand;
	processingDone :PartTrackingProcssingDoneCommand;
END_VAR

(*

## Short summary

This abstract property returns the class name of the concrete object, 
which is useful for logging/debugging purpose or to check the class name
for ``__DELETE`` in factories (sometimes it's necessary to do more 
than just to free the memory).

.. <legal notes>

legal notes
=================
| SPDX-FileCopyrightText: © 2022 ekvip automation GmbH <info@ekvip.de>
| SPDX-License-Identifier: Apache-2.0
| For details check: Apache-2.0_

.. _Apache-2.0: https://www.apache.org/licenses/LICENSE-2.0

.. </legal notes>

*)

PROPERTY className : CNM_AbstractObject.ClassName
GET
 className := 'CNM_ProductionMetrics.PartTrackingCommands';
END_GET
END_PROPERTY

(*

## Short summary

This command creates a part counter dataset for the currenttly processed part.
The part will be counted as OK part if the nokReason is set to 0 and not OK otherwise.
The additionalMessage can be used to provide additional information, e.g. SPC part or measurements that are out of the permissible range. 

.. <legal notes>

legal notes
=================
| SPDX-FileCopyrightText: © 2025 ekvip automation GmbH <info@ekvip.de>
| SPDX-License-Identifier: Apache-2.0
| For details check: Apache-2.0_

.. _Apache-2.0: https://www.apache.org/licenses/LICENSE-2.0

.. </legal notes>

*)
METHOD partProcessingDone : CNM_CommandInterfaces.ISingleAttempt
VAR_INPUT
	(* the part number as string *)
	partIdentifier	: Tc2_System.T_MaxString;
	(* if not 0, the record will be marked as not OK part *)
	nokReason	: DWORD;
	(* can be used to provide additional informations for the record, e.g. voltage too low *)
	additionalMessage	: Tc2_System.T_MaxString;
END_VAR
THIS^.processingDone.setParameters(
	partIdentifier := partIdentifier,
	nokReason := nokReason,
	additionalMessage := additionalMessage
);
partProcessingDone := THIS^.processingDone;
END_METHOD

(*

## Short summary

This command starts a new process cycle and sets the start time stamp for the corresponding partIdentifier.

**Attention:** calling this method clears the currently set part data, e.g. if the last process cycle couldn't be finished.

.. <legal notes>

legal notes
=================
| SPDX-FileCopyrightText: © 2025 ekvip automation GmbH <info@ekvip.de>
| SPDX-License-Identifier: Apache-2.0
| For details check: Apache-2.0_

.. _Apache-2.0: https://www.apache.org/licenses/LICENSE-2.0

.. </legal notes>

*)
METHOD partProcessingStarted : CNM_CommandInterfaces.ISingleAttempt
VAR_INPUT
	(* the part number as string *)
	partIdentifier	: Tc2_System.T_MaxString;
END_VAR
THIS^.startProcessing.setParameters(
	partIdentifier := partIdentifier
);
partProcessingStarted := THIS^.startProcessing;
END_METHOD

METHOD INTERNAL setRecorder : BOOL
VAR_INPUT
	recorder :CNM_ProductionMetricInterfaces.IPartTracker;
END_VAR
IF THIS^.isObjectValid(recorder) THEN
	THIS^.startProcessing.setRecorder(recorder);
	THIS^.processingDone.setRecorder(recorder);
END_IF
END_METHOD

END_FUNCTION_BLOCK

// ---- classes/Measurements/PartTracking/Commands/PartTrackingProcssingStartedCommand.TcPOU
(*
## Short summary

This command starts a new process cycle and sets the start time stamp for the corresponding partIdentifier.

**Attention:** calling this method clears the currently set part data, e.g. if the last process cycle couldn't be finished.

.. <legal notes>

legal notes
=================
| SPDX-FileCopyrightText: © 2025 ekvip automation GmbH <info@ekvip.de>
| SPDX-License-Identifier: Apache-2.0
| For details check: Apache-2.0_

.. _Apache-2.0: https://www.apache.org/licenses/LICENSE-2.0

.. </legal notes>

*)
FUNCTION_BLOCK PartTrackingProcssingStartedCommand EXTENDS CNM_AbstractObject.Object IMPLEMENTS CNM_CommandInterfaces.ISingleAttempt
VAR
	recorder :CNM_ProductionMetricInterfaces.IPartTracker;
	partIdentifier :Tc2_System.T_MaxString;
END_VAR

(*

## Short summary

This abstract property returns the class name of the concrete object, 
which is useful for logging/debugging purpose or to check the class name
for ``__DELETE`` in factories (sometimes it's necessary to do more 
than just to free the memory).

.. <legal notes>

legal notes
=================
| SPDX-FileCopyrightText: © 2022 ekvip automation GmbH <info@ekvip.de>
| SPDX-License-Identifier: Apache-2.0
| For details check: Apache-2.0_

.. _Apache-2.0: https://www.apache.org/licenses/LICENSE-2.0

.. </legal notes>

*)
PROPERTY className : CNM_AbstractObject.ClassName
GET
className := 'CNM_ProductionMetrics.PartTrackingProcssingStartedCommand';
END_GET
END_PROPERTY

(*

## Short summary

Invokes the action associated with this interface.

.. <legal notes>

legal notes
=================
| SPDX-FileCopyrightText: © 2024 ekvip automation GmbH <info@ekvip.de>
| SPDX-License-Identifier: Apache-2.0
| For details check: Apache-2.0_

.. _Apache-2.0: https://www.apache.org/licenses/LICENSE-2.0

.. </legal notes>



*)
METHOD invoke : CNM_ReturnTypes.SingleExecutionResult
IF THIS^.isObjectValid(THIS^.recorder) THEN
	invoke := THIS^.recorder.setPartProcessingStarted(
		partIdentifier := THIS^.partIdentifier
	);
ELSE
	invoke := CNM_ReturnTypes.SingleExecutionResult.ABORTED;
END_IF
END_METHOD

METHOD INTERNAL setParameters
VAR_INPUT
	(* the part number as string *)
	partIdentifier :Tc2_System.T_MaxString;
END_VAR
THIS^.partIdentifier := partIdentifier;
END_METHOD

(*
## Short summary

This methods sets the parttracking recorder interface on which the command is executed.

.. <legal notes>

legal notes
=================
| SPDX-FileCopyrightText: © 2025 ekvip automation GmbH <info@ekvip.de>
| SPDX-License-Identifier: Apache-2.0
| For details check: Apache-2.0_

.. _Apache-2.0: https://www.apache.org/licenses/LICENSE-2.0

.. </legal notes>

*)

METHOD INTERNAL setRecorder
VAR_INPUT
	recorder :CNM_ProductionMetricInterfaces.IPartTracker;
END_VAR
IF THIS^.isObjectValid(recorder) THEN
	THIS^.recorder := recorder;
END_IF
END_METHOD

END_FUNCTION_BLOCK

// ---- classes/Measurements/PartTracking/Commands/PartTrackingProcssingDoneCommand.TcPOU
(*
## Short summary

This command starts a new process cycle and sets the start time stamp for the corresponding partIdentifier.

**Attention:** calling this method clears the currently set part data, e.g. if the last process cycle couldn't be finished.

.. <legal notes>

legal notes
=================
| SPDX-FileCopyrightText: © 2025 ekvip automation GmbH <info@ekvip.de>
| SPDX-License-Identifier: Apache-2.0
| For details check: Apache-2.0_

.. _Apache-2.0: https://www.apache.org/licenses/LICENSE-2.0

.. </legal notes>

*)
FUNCTION_BLOCK PartTrackingProcssingDoneCommand EXTENDS CNM_AbstractObject.Object IMPLEMENTS CNM_CommandInterfaces.ISingleAttempt
VAR
	recorder :CNM_ProductionMetricInterfaces.IPartTracker;
	(* the part number as string *)
	partIdentifier :Tc2_System.T_MaxString;
	(* if not 0, the record will be marked as not OK part *)
	nokReason :DWORD;
	(* can be used to provide additional informations for the record, e.g. voltage too low *)
	additionalMessage :Tc2_System.T_MaxString;
END_VAR

(*

## Short summary

This abstract property returns the class name of the concrete object, 
which is useful for logging/debugging purpose or to check the class name
for ``__DELETE`` in factories (sometimes it's necessary to do more 
than just to free the memory).

.. <legal notes>

legal notes
=================
| SPDX-FileCopyrightText: © 2022 ekvip automation GmbH <info@ekvip.de>
| SPDX-License-Identifier: Apache-2.0
| For details check: Apache-2.0_

.. _Apache-2.0: https://www.apache.org/licenses/LICENSE-2.0

.. </legal notes>

*)
PROPERTY className : CNM_AbstractObject.ClassName
GET
className := 'CNM_ProductionMetrics.PartTrackingProcssingDoneCommand';
END_GET
END_PROPERTY

(*

## Short summary

Invokes the action associated with this interface.

.. <legal notes>

legal notes
=================
| SPDX-FileCopyrightText: © 2024 ekvip automation GmbH <info@ekvip.de>
| SPDX-License-Identifier: Apache-2.0
| For details check: Apache-2.0_

.. _Apache-2.0: https://www.apache.org/licenses/LICENSE-2.0

.. </legal notes>



*)
METHOD invoke : CNM_ReturnTypes.SingleExecutionResult
IF THIS^.isObjectValid(THIS^.recorder) THEN
	invoke := THIS^.recorder.setPartProcessingDone(
		partIdentifier := THIS^.partIdentifier,
		nokReason := THIS^.nokReason,
		additionalMessage := THIS^.additionalMessage
	);
ELSE
	invoke := CNM_ReturnTypes.SingleExecutionResult.ABORTED;
END_IF
END_METHOD

METHOD INTERNAL setParameters
VAR_INPUT
	(* the part number as string *)
	partIdentifier :Tc2_System.T_MaxString;
		(* if not 0, the record will be marked as not OK part *)
	nokReason :DWORD;
	(* can be used to provide additional informations for the record, e.g. voltage too low *)
	additionalMessage :Tc2_System.T_MaxString;
END_VAR
THIS^.partIdentifier := partIdentifier;
THIS^.nokReason := nokReason;
THIS^.additionalMessage := additionalMessage;
END_METHOD

(*
## Short summary

This methods sets the parttracking recorder interface on which the command is executed.

.. <legal notes>

legal notes
=================
| SPDX-FileCopyrightText: © 2025 ekvip automation GmbH <info@ekvip.de>
| SPDX-License-Identifier: Apache-2.0
| For details check: Apache-2.0_

.. _Apache-2.0: https://www.apache.org/licenses/LICENSE-2.0

.. </legal notes>

*)

METHOD INTERNAL setRecorder
VAR_INPUT
	recorder :CNM_ProductionMetricInterfaces.IPartTracker;
END_VAR
IF THIS^.isObjectValid(recorder) THEN
	THIS^.recorder := recorder;
END_IF
END_METHOD

END_FUNCTION_BLOCK

// ---- classes/Measurements/PartTracking/PartTrackingConfiguration.TcPOU
(* 
## Short summary

This class is a data transfer object for configurable part data attributes. 
It is intended to be uses within a fluid configuration interface. 

.. <legal notes>

legal notes
=================
| SPDX-FileCopyrightText: © 2025 ekvip automation GmbH <info@ekvip.de>
| SPDX-License-Identifier: Apache-2.0
| For details check: Apache-2.0_

.. _Apache-2.0: https://www.apache.org/licenses/LICENSE-2.0

.. </legal notes>

*)

FUNCTION_BLOCK PartTrackingConfiguration EXTENDS CycleTimeRecorderConfiguration IMPLEMENTS CNM_ProductionMetricInterfaces.IPartTrackerConfiguration
VAR
	configuredOrder :Tc2_System.T_MaxString;
END_VAR

(*

## Short summary

This abstract property returns the class name of the concrete object, 
which is useful for logging/debugging purpose or to check the class name
for ``__DELETE`` in factories (sometimes it's necessary to do more 
than just to free the memory).

.. <legal notes>

legal notes
=================
| SPDX-FileCopyrightText: © 2022 ekvip automation GmbH <info@ekvip.de>
| SPDX-License-Identifier: Apache-2.0
| For details check: Apache-2.0_

.. _Apache-2.0: https://www.apache.org/licenses/LICENSE-2.0

.. </legal notes>

*)
PROPERTY className : CNM_AbstractObject.ClassName
GET
className := 'PartCounterConfiguration';
END_GET
END_PROPERTY

(* 
## Short summary

This property can be used to set and read the current batch number as string.
The batch number will be written into every measurement entry.

.. <legal notes>

legal notes
=================
| SPDX-FileCopyrightText: © 2025 ekvip automation GmbH <info@ekvip.de>
| SPDX-License-Identifier: Apache-2.0
| For details check: Apache-2.0_

.. _Apache-2.0: https://www.apache.org/licenses/LICENSE-2.0

.. </legal notes>

*)
PROPERTY order : Tc2_System.T_MaxString
GET
order := THIS^.configuredOrder;
END_GET
SET
THIS^.configuredOrder := order;
END_SET
END_PROPERTY

END_FUNCTION_BLOCK

// ---- classes/Measurements/PartTracking/PartTrackingRecorder.TcPOU
FUNCTION_BLOCK PartTrackingRecorder EXTENDS CNM_OpModeHandler.AbstractCyclicNode IMPLEMENTS CNM_ProductionMetricInterfaces.IPartTracker
VAR
	currentData :CNM_ProductionMetricInterfaces.PartDataTrackingStruct;
	(* queue for the measurements *)
	dataSetList :CNM_Collections.LinkedList;
	(* the variable that is used to provide data for the database *)
	{ attribute 'TcHmiSymbol.ShowRecursively' }
	partDataSet :CNM_ProductionMetricInterfaces.PartDataTrackingStruct;
	(* mailbox flag for the database that we have a new entry, should be reset by the server when data was read *)
	{ attribute 'TcHmiSymbol.Show' }
	newDataAvailable :BOOL := FALSE;
	(* command delegates *)
	partTrackerCommands :PartTrackingCommands;
	(* error for failed queryInterface *)
	interfaceQueryFailedAlarm :CNM_ConcreteMessages.TcError(event := Global.TC_EVENTS.MemoryErrors.PartTrackerQueryInterfacFailed , injectedService := THIS^.messageService);
	(* error for maximum queue size *)
	maxQueueSizeAlarm :CNM_ConcreteMessages.TcError(event := Global.TC_EVENTS.MemoryErrors.PartTrackingMaxQueueSize, injectedService := THIS^.messageService); 
END_VAR

(*

## Short summary

This abstract property returns the class name of the concrete object, 
which is useful for logging/debugging purpose or to check the class name
for ``__DELETE`` in factories (sometimes it's necessary to do more 
than just to free the memory).

.. <legal notes>

legal notes
=================
| SPDX-FileCopyrightText: © 2022 ekvip automation GmbH <info@ekvip.de>
| SPDX-License-Identifier: Apache-2.0
| For details check: Apache-2.0_

.. _Apache-2.0: https://www.apache.org/licenses/LICENSE-2.0

.. </legal notes>

*)
PROPERTY className : CNM_AbstractObject.ClassName
GET
className := 'PartTrackingRecorder';
END_GET
END_PROPERTY

(* 
## Short summary

This property is a fluent interface that provides single attempt commands, which can be evaluated by a cycle manager instance.
### Example 
```
	
	// execute command when leaving a step 
	cycleManager.leave(
		partTracker.commands.partProcessingDone(
			partIdentifier := 'Part123',
			nokReason := 0,
			additionalMessage := 'SPC Part'
		)
	);  
```	

.. <legal notes>

legal notes
=================
| SPDX-FileCopyrightText: © 2025 ekvip automation GmbH <info@ekvip.de>
| SPDX-License-Identifier: Apache-2.0
| For details check: Apache-2.0_

.. _Apache-2.0: https://www.apache.org/licenses/LICENSE-2.0

.. </legal notes>
	
*)

PROPERTY commands : CNM_ProductionMetricInterfaces.IPartTrackingRecorderCommands
GET
commands := THIS^.partTrackerCommands;
END_GET
END_PROPERTY

(*

## Short summary

This property returns an fluent interface for part counter configuration.
The following things should be configured after a type / product / batch change was performed:
 -batch: insert the current/new batch name/number as string
 -product type: either the name of the overall product or the individual feed parts to be processed

The process name can be set once during the initialization of the PLC as it usually doesn't change.

.. <legal notes>

legal notes
=================
| SPDX-FileCopyrightText: © 2025 ekvip automation GmbH <info@ekvip.de>
| SPDX-License-Identifier: Apache-2.0
| For details check: Apache-2.0_

.. _Apache-2.0: https://www.apache.org/licenses/LICENSE-2.0

.. </legal notes>

*)
PROPERTY configuration : CNM_ProductionMetricInterfaces.IPartTrackerConfiguration
GET
VAR_INST
	config :PartTrackingConfiguration;
END_VAR
configuration := config;
END_GET
END_PROPERTY

(* 
## Short summary

This method disables a node (E.g. axes should be disabled). It can take mutliple cycles. It has to be implemented for every node/device.
The execute input needs a rising edge to execute the method.
If there is nothing to disable, just return a 'SUCCESS' state.

This method is called automatically by the operation mode handler.

.. <legal notes>

legal notes
=================
| SPDX-FileCopyrightText: © 2024 ekvip automation GmbH <info@ekvip.de>
| SPDX-License-Identifier: Apache-2.0
| For details check: Apache-2.0_

.. _Apache-2.0: https://www.apache.org/licenses/LICENSE-2.0

.. </legal notes>

*)
METHOD disable : CNM_ReturnTypes.SingleExecutionState
VAR_INPUT
	execute	: BOOL;
END_VAR
// nothing to disable
disable := CNM_ReturnTypes.SingleExecutionState.SUCCESS;
END_METHOD

(* 
## Short summary

This method enables a node. It can take mutliple cycles. It has to be implemented for every node/device.
The intention is to enable devices here, e.g. axes, laser, dispenser etc.
The execute input needs a rising edge to execute the method.
If there is nothing to enable, just return a 'SUCCESS' state.

This method is called automatically by the operation mode handler.

.. <legal notes>

legal notes
=================
| SPDX-FileCopyrightText: © 2024 ekvip automation GmbH <info@ekvip.de>
| SPDX-License-Identifier: Apache-2.0
| For details check: Apache-2.0_

.. _Apache-2.0: https://www.apache.org/licenses/LICENSE-2.0

.. </legal notes>

*)
METHOD enable : CNM_ReturnTypes.SingleExecutionState
VAR_INPUT
	execute	: BOOL;
END_VAR
// nothing to enable
enable := CNM_ReturnTypes.SingleExecutionState.SUCCESS;
END_METHOD

(*

## Short summary

The constructor ``FB_init`` is needed to create an unique hash code.
The hash code is a pseudo random number create with a [xorshift](https://en.wikipedia.org/wiki/Xorshift) algorithm.
It can be overwritten on derivations, because it will be called implicit, ``SUPER^.FB_init()`` is not required.
For more information check: [Behavoir with derived function blocks](https://infosys.beckhoff.com/content/1033/tc3_plc_intro/5482088715.html?id=6983869892358031022)

.. <legal notes>

legal notes
=================
| SPDX-FileCopyrightText: © 2022 ekvip automation GmbH <info@ekvip.de>
| SPDX-License-Identifier: Apache-2.0
| For details check: Apache-2.0_

.. _Apache-2.0: https://www.apache.org/licenses/LICENSE-2.0

.. </legal notes>



*)
METHOD FB_init : BOOL
VAR_INPUT
	(* if TRUE, the retain variables are initialized (warm start / cold start)*)
	bInitRetains	: BOOL;
	(* if TRUE, the instance afterwards gets moved into the copy code (online change) *)
	bInCopyCode	:BOOL;
	(* the node were this node should be appended to *)
	parentNode :CNM_OpModeHandler.INodeInitialization;
END_VAR
THIS^.hmiInfo.template := 'PartTrackingRecorder';
THIS^.isInHome := TRUE;
END_METHOD

(* 
## Short summary

This method contains instructions and sequences for the init mode. 
This mode is intended for initializing a machine, e.g. loading product type data from recipes, establish a connection to global production systems (MES).
If the node should do nothing, return a 'SUCCESS'.
It should run until all initializations are done or the mode is stopped immedtiately or a stop request is raised (THIS^.modeControl.stopRequest). 
This method is called automatically by the operation mode handler.

**Attention:** If this method returns the state 'ERROR', the operation mode handler automatically disables the whole machine! 

.. <legal notes>

legal notes
=================
| SPDX-FileCopyrightText: © 2024 ekvip automation GmbH <info@ekvip.de>
| SPDX-License-Identifier: Apache-2.0
| For details check: Apache-2.0_

.. _Apache-2.0: https://www.apache.org/licenses/LICENSE-2.0

.. </legal notes>

*)
METHOD initialize : CNM_ReturnTypes.SingleExecutionState
VAR_INPUT
	execute	: BOOL;
END_VAR
THIS^.partTrackerCommands.setRecorder(THIS^);
initialize := CNM_ReturnTypes.SingleExecutionState.SUCCESS;
END_METHOD

(*
## Short summary

This property getter returns the maximum queue size for the data recorder. 
If the dataset list has reached this size, no other dataset will be stored and an alarm will be raised.
For this class the maximum queue size can be configured as library parameter ''QUEUE_SIZE_FOR_DATA_RECORDS_PER_RECORDER''.
Overwrite this property for extended classes as the default implementation accesses the Parameter List of the CNM_ProductionMetrics library! 

.. <legal notes>

legal notes
=================
| SPDX-FileCopyrightText: © 2022 ekvip automation GmbH <info@ekvip.de>
| SPDX-License-Identifier: Apache-2.0
| For details check: Apache-2.0_

.. _Apache-2.0: https://www.apache.org/licenses/LICENSE-2.0

.. </legal notes>

*)

PROPERTY PROTECTED maxQueueSize : UDINT
GET
maxQueueSize := Settings.QUEUE_SIZE_FOR_DATA_RECORDS_PER_RECORDER;
END_GET
END_PROPERTY

(* 
## Short summary

This method will be called in every cycle for a node. It can be used to implement hardware drivers/measurements/monitoring.
The returned state defines the overall state of the node. It should return BUSY when the node executes a command, otherwise SUCCESS( or IDLE if there is nothing to do). 
(Simple monitoring is not a command an should return SUCCESS).  


**Attention:** the returned SingleExecutionState will be evaluated cyclically wihtin the node tree. 
In case a node returns an ERROR state, the whole machine will be disabled. 
Return ERROR only for fatal or critical errors and handle other errors within the node.
 

.. <legal notes>

legal notes
=================
| SPDX-FileCopyrightText: © 2025 ekvip automation GmbH <info@ekvip.de>
| SPDX-License-Identifier: Apache-2.0
| For details check: Apache-2.0_

.. _Apache-2.0: https://www.apache.org/licenses/LICENSE-2.0

.. </legal notes>
	
*)
METHOD run : CNM_ReturnTypes.SingleExecutionState
VAR_INST
	cycleManager :CNM_CycleManager.SimpleCycleManager;
END_VAR
VAR CONSTANT
	WAIT_FOR_DATA :DINT := 10;
	SET_DATA :DINT := 11;
	DATA_ERROR :DINT := 12;
	WAIT_DATA_RECEIVED :DINT := 13;
END_VAR
VAR
	data :CNM_ProductionMetricInterfaces.IPartTrackingData;
END_VAR
cycleManager(execute := TRUE);

CASE cycleManager.step.current OF
CNM_ReturnTypes.DefaultSteps.STEP.INIT:
	run := CNM_ReturnTypes.SingleExecutionState.SUCCESS;
	cycleManager.proceedWith(WAIT_FOR_DATA);
WAIT_FOR_DATA:
	run := CNM_ReturnTypes.SingleExecutionState.SUCCESS;
	IF (THIS^.dataSetList.size > 0) THEN
		run := CNM_ReturnTypes.SingleExecutionState.BUSY;
		cycleManager.proceedWith(SET_DATA); 
	END_IF
SET_DATA:
	run := CNM_ReturnTypes.SingleExecutionState.BUSY;
	IF (__QUERYINTERFACE(THIS^.dataSetList.dequeue(), data)) THEN
		(* fill dataslot *)
		THIS^.partDataSet := data.dataset;
		(* delete DTO *)
		data.destruct();
		(* set mailbox flag *)
		THIS^.newDataAvailable := TRUE;
		cycleManager.proceedWith(WAIT_DATA_RECEIVED);
	ELSE
		cycleManager.proceedWith(DATA_ERROR);
	END_IF
DATA_ERROR:
	cycleManager.step.next := SET_DATA;
	cycleManager.handle(THIS^.interfaceQueryFailedAlarm);
WAIT_DATA_RECEIVED:
	run := CNM_ReturnTypes.SingleExecutionState.BUSY;
	IF (NOT THIS^.newDataAvailable) THEN
		// clear data slot
		Tc2_System.MEMSET(destAddr := ADR(THIS^.partDataSet), 0, SIZEOF(THIS^.partDataSet));
		run := CNM_ReturnTypes.SingleExecutionState.SUCCESS;
		cycleManager.proceedWith(WAIT_FOR_DATA);
	END_IF
END_CASE
END_METHOD

(*

## Short summary

This method creates a part counter dataset for the currenttly processed part.
The part will be counted as OK part if the nokReason is set to 0 and not OK otherwise.
The additionalMessage can be used to provide additional information, e.g. SPC part or measurements that are out of the permissible range. 

.. <legal notes>

legal notes
=================
| SPDX-FileCopyrightText: © 2025 ekvip automation GmbH <info@ekvip.de>
| SPDX-License-Identifier: Apache-2.0
| For details check: Apache-2.0_

.. _Apache-2.0: https://www.apache.org/licenses/LICENSE-2.0

.. </legal notes>

*)
METHOD setPartProcessingDone : CNM_ProductionMetricInterfaces.CNM_ReturnTypes.SingleExecutionResult
VAR_INPUT
	(* the part number as string *)
	partIdentifier	: Tc2_System.T_MaxString;
	(* if not 0, the record will be marked as not OK part *)
	nokReason	: DWORD;
	(* can be used to provide additional informations for the record, e.g. voltage too low *)
	additionalMessage	: Tc2_System.T_MaxString;
END_VAR
VAR
	dto :POINTER TO PartTrackingData;
	backupEndTimestamp :LDT;
END_VAR
setPartProcessingDone := CNM_ReturnTypes.SingleExecutionResult.ABORTED;
// check if we can queue the dataset - throw error if the max queuesize is reached
IF ( THIS^.dataSetList.size >= THIS^.maxQueueSize ) THEN
	THIS^.maxQueueSizeAlarm.throw();
	RETURN;
END_IF

backupEndTimestamp  := THIS^.currentData.endTimestamp;

THIS^.currentData.partIdentifier := partIdentifier;
THIS^.currentData.cycleTime := 
	SEL(
		TO_UDINT(THIS^.currentData.endTimestamp) > 0, 
		TO_LTIME(0), 
		TO_LTIME(GetCurrentLTimeStamp() - THIS^.currentData.endTimestamp )
	);
THIS^.currentData.endTimestamp := GetCurrentLTimeStamp();
THIS^.currentData.processingTime := 
	SEL(
		TO_UDINT(THIS^.currentData.startTimestamp) > 0, 
		TO_LTIME(0), 
		TO_LTIME(THIS^.currentData.endTimestamp - THIS^.currentData.startTimestamp));
THIS^.currentData.process := THIS^.configuration.process;
THIS^.currentData.productType := THIS^.configuration.productType;
THIS^.currentData.targetCycletime := THIS^.configuration.targetCycleTime;
THIS^.currentData.additionalMessage := additionalMessage;
THIS^.currentData.nokReason := nokReason;
THIS^.currentData.order := THIS^.configuration.order;
dto := __NEW(PartTrackingData(data := THIS^.currentData));
IF (dto <> 0) THEN
	setPartProcessingDone := THIS^.dataSetList.append(dto^);
ELSE
	// restore data for retry
	THIS^.currentData.endTimestamp := backupEndTimestamp;
END_IF
END_METHOD

(*

## Short summary

This method starts a new process cycle and sets the start time stamp for the corresponding partIdentifier.

**Attention:** calling this method clears the currently set part data, e.g. if the last process cycle couldn't be finished.

.. <legal notes>

legal notes
=================
| SPDX-FileCopyrightText: © 2025 ekvip automation GmbH <info@ekvip.de>
| SPDX-License-Identifier: Apache-2.0
| For details check: Apache-2.0_

.. _Apache-2.0: https://www.apache.org/licenses/LICENSE-2.0

.. </legal notes>

*)
METHOD setPartProcessingStarted : CNM_ProductionMetricInterfaces.CNM_ReturnTypes.SingleExecutionResult
VAR_INPUT
	(* the part number as string *)
	partIdentifier	: Tc2_System.T_MaxString;
END_VAR
THIS^.currentData.partIdentifier := partIdentifier;
THIS^.currentData.startTimestamp := GetCurrentLTimeStamp();
setPartProcessingStarted := CNM_ReturnTypes.SingleExecutionResult.SUCCESS;
END_METHOD

(* 
## Short summary

This method executes stops all movements of a node. It has to be overwritten for every node. 
E.g. axes should perform a quickstop, cylinders should be turned off, etc.
If the node should do nothing, return a 'SUCCESS'.
It should stop axes/cylinders/process (e.g. laser welding, dispensing) endless until the manual mode is stopped via stop request or immediate stop.
This method is called automatically by the operation mode handler before disabling the machine or if the operator selects an immediate stop.

**Attention:** If this method returns the state 'ERROR', the operation mode handler automatically disables the whole machine! 

.. <legal notes>

legal notes
=================
| SPDX-FileCopyrightText: © 2024 ekvip automation GmbH <info@ekvip.de>
| SPDX-License-Identifier: Apache-2.0
| For details check: Apache-2.0_

.. _Apache-2.0: https://www.apache.org/licenses/LICENSE-2.0

.. </legal notes>

*)
METHOD stopImmediate : CNM_ReturnTypes.SingleExecutionState
VAR_INPUT
	execute	: BOOL;
END_VAR
// nothing to stop
stopImmediate := CNM_ReturnTypes.SingleExecutionState.SUCCESS;
END_METHOD

END_FUNCTION_BLOCK

// ---- classes/Measurements/SimpleMeasurement/commands/MeasurementAddEntryCommand.TcPOU
(*
## Short summary

This command can be used to create and store a new measurement data set.

.. <legal notes>

legal notes
=================
| SPDX-FileCopyrightText: © 2025 ekvip automation GmbH <info@ekvip.de>
| SPDX-License-Identifier: Apache-2.0
| For details check: Apache-2.0_

.. _Apache-2.0: https://www.apache.org/licenses/LICENSE-2.0

.. </legal notes>

*)
FUNCTION_BLOCK MeasurementAddEntryCommand EXTENDS CNM_AbstractObject.Object IMPLEMENTS CNM_CommandInterfaces.ISingleAttempt
VAR
	recorder :CNM_ProductionMetricInterfaces.IMeasurementRecorder;
	(* product identifier for that specific part *)
	partIdentifier	:Tc2_System.T_MaxString;
	(* name of the measurement, e.g. label position, cell voltage, oven temperature *)
	nameMeasurement	: Tc2_System.T_MaxString;
	(* unit of the measurement, e.g. mm, V, °C *)
	unit	: CNM_ProductionMetricInterfaces.UnitString;
	(* Permissible value range of the measurement for OK parts*)
	range	: CNM_ProductionMetricInterfaces.MeasurementRangeStruct;
	(* value of the measurement *)
	value	: LREAL;
END_VAR

(*

## Short summary

This abstract property returns the class name of the concrete object, 
which is useful for logging/debugging purpose or to check the class name
for ``__DELETE`` in factories (sometimes it's necessary to do more 
than just to free the memory).

.. <legal notes>

legal notes
=================
| SPDX-FileCopyrightText: © 2022 ekvip automation GmbH <info@ekvip.de>
| SPDX-License-Identifier: Apache-2.0
| For details check: Apache-2.0_

.. _Apache-2.0: https://www.apache.org/licenses/LICENSE-2.0

.. </legal notes>

*)
PROPERTY className : CNM_AbstractObject.ClassName
GET
className := 'CNM_ProductionMetrics.CycleTimeStartCycleCommand';
END_GET
END_PROPERTY

(*

## Short summary

Invokes the action associated with this interface.

.. <legal notes>

legal notes
=================
| SPDX-FileCopyrightText: © 2024 ekvip automation GmbH <info@ekvip.de>
| SPDX-License-Identifier: Apache-2.0
| For details check: Apache-2.0_

.. _Apache-2.0: https://www.apache.org/licenses/LICENSE-2.0

.. </legal notes>



*)
METHOD invoke : CNM_ReturnTypes.SingleExecutionResult
IF THIS^.isObjectValid(THIS^.recorder) THEN
	invoke := THIS^.recorder.addMeasurementEntry(
		partIdentifier := THIS^.partIdentifier,
		name := THIS^.nameMeasurement,
		unit := THIS^.unit,
		range := THIS^.range,
		value := THIS^.value
	);
ELSE
	invoke := CNM_ReturnTypes.SingleExecutionResult.ABORTED;
END_IF
END_METHOD

METHOD INTERNAL setParameters
VAR_INPUT
	(* product identifier for that specific part *)
	partIdentifier	:Tc2_System.T_MaxString;
	(* name of the measurement, e.g. label position, cell voltage, oven temperature *)
	name	: Tc2_System.T_MaxString;
	(* unit of the measurement, e.g. mm, V, °C *)
	unit	: CNM_ProductionMetricInterfaces.UnitString;
	(* Permissible value range of the measurement for OK parts*)
	range	: CNM_ProductionMetricInterfaces.MeasurementRangeStruct;
	(* value of the measurement *)
	value	: LREAL;
END_VAR
THIS^.partIdentifier := partIdentifier;
THIS^.nameMeasurement := name;
THIS^.unit := unit;
THIS^.range := range;
THIS^.value := value;
END_METHOD

(*
## Short summary

This methods sets the cycletime recorder interface on which the command is executed.

.. <legal notes>

legal notes
=================
| SPDX-FileCopyrightText: © 2025 ekvip automation GmbH <info@ekvip.de>
| SPDX-License-Identifier: Apache-2.0
| For details check: Apache-2.0_

.. _Apache-2.0: https://www.apache.org/licenses/LICENSE-2.0

.. </legal notes>

*)

METHOD setRecorder
VAR_INPUT
	recorder :CNM_ProductionMetricInterfaces.IMeasurementRecorder;
END_VAR
IF THIS^.isObjectValid(recorder) THEN
	THIS^.recorder := recorder;
END_IF
END_METHOD

END_FUNCTION_BLOCK

// ---- classes/Measurements/SimpleMeasurement/commands/MeasurementRecorderCommands.TcPOU
(* 
## Short summary

This class is a collection of cycle time recorder commands that provides a fluent interface that provides single attempt commands, which can be evaluated by a cycle manager instance.
### Example 
```
	
	// execute command when leaving a step 
	cycleManager.leave(
		measurement.commands.addMeasurementEntry(
			partIdentifier	:= 'Part123',
			name := 'Voltage Check',
			unit := 'V',
			range := productType.VoltageCheck.Range,
			value := 3.14
		)
	); 
```	

.. <legal notes>

legal notes
=================
| SPDX-FileCopyrightText: © 2025 ekvip automation GmbH <info@ekvip.de>
| SPDX-License-Identifier: Apache-2.0
| For details check: Apache-2.0_

.. _Apache-2.0: https://www.apache.org/licenses/LICENSE-2.0

.. </legal notes>
	
*)

FUNCTION_BLOCK MeasurementRecorderCommands EXTENDS CNM_AbstractObject.Object IMPLEMENTS CNM_ProductionMetricInterfaces.IMeasurementRecorderCommands
VAR
	addMeasurementCommand :MeasurementAddEntryCommand;
END_VAR

(*
## Short summary

This command creates a new measurement entry and queues it for the database insection.

.. <legal notes>

legal notes
=================
| SPDX-FileCopyrightText: © 2025 ekvip automation GmbH <info@ekvip.de>
| SPDX-License-Identifier: Apache-2.0
| For details check: Apache-2.0_

.. _Apache-2.0: https://www.apache.org/licenses/LICENSE-2.0

.. </legal notes>

*)
METHOD addMeasurement : CNM_CommandInterfaces.ISingleAttempt
VAR_INPUT
	(* product identifier for that specific part *)
	partIdentifier	: Tc2_System.T_MaxString;
	(* name of the measurement, e.g. label position, cell voltage, oven temperature *)
	name	: Tc2_System.T_MaxString;
	(* unit of the measurement, e.g. mm, V, °C *)
	unit	: CNM_ProductionMetricInterfaces.UnitString;
	(* Permissible value range of the measurement for OK parts*)
	range	: CNM_ProductionMetricInterfaces.MeasurementRangeStruct;
	(* value of the measurement *)
	value	: LREAL;
END_VAR
THIS^.addMeasurementCommand.setParameters(
	partIdentifier := partIdentifier,
	name := name,
	unit := unit,
	range := range,
	value := value 
);
addMeasurement := THIS^.addMeasurementCommand;
END_METHOD

(*

## Short summary

This abstract property returns the class name of the concrete object, 
which is useful for debugging purpose or to check the class name for 
``__DELETE`` in factories (sometimes it's necessary to do more 
than just to free the memory).

**Attention:**: 
	For derivations: **It is necessary that this property is overridden by the concrete class**

.. <legal notes>

legal notes
=================
| SPDX-FileCopyrightText: © 2022 ekvip automation GmbH <info@ekvip.de>
| SPDX-License-Identifier: Apache-2.0
| For details check: Apache-2.0_

.. _Apache-2.0: https://www.apache.org/licenses/LICENSE-2.0

.. </legal notes>

*)

PROPERTY className : CNM_AbstractObject.ClassName
GET
 className := 'CNM_ProductionMetrics.MeasurementRecorderCommands';
END_GET
END_PROPERTY

METHOD INTERNAL setRecorder : BOOL
VAR_INPUT
	recorder :CNM_ProductionMetricInterfaces.IMeasurementRecorder;
END_VAR
IF THIS^.isObjectValid(recorder) THEN
	THIS^.addMeasurementCommand.setRecorder(recorder);
END_IF
END_METHOD

END_FUNCTION_BLOCK

// ---- classes/Measurements/SimpleMeasurement/MeasurementRecorder.TcPOU
(*
## Short summary


This is class that can be used to generate process related measurements and store them to a Database.
Measurements are going to be queued in a linked list and send to the database one after another. 

.. <legal notes>

legal notes
=================
| SPDX-FileCopyrightText: © 2025 ekvip automation GmbH <info@ekvip.de>
| SPDX-License-Identifier: Apache-2.0
| For details check: Apache-2.0_

.. _Apache-2.0: https://www.apache.org/licenses/LICENSE-2.0

.. </legal notes>

*)

FUNCTION_BLOCK MeasurementRecorder EXTENDS CNM_OpModeHandler.AbstractCyclicNode 
	IMPLEMENTS 	CNM_ProductionMetricInterfaces.IMeasurementRecorder
VAR
	(* queue for the measurements *)
	dataSetList :CNM_Collections.LinkedList;
	(* the variable that is used to provide data for the database *)
	{ attribute 'TcHmiSymbol.ShowRecursively' }
	measurement :CNM_ProductionMetricInterfaces.MeasurementEntryStruct;
	(* mailbox flag for the database that we have a new entry, should be reset by the server when data was read *)
	{ attribute 'TcHmiSymbol.Show' }
	newDataAvailable :BOOL := FALSE;
	(* command delegates *)
	measurementCommands :MeasurementRecorderCommands;
	(* error for failed queryInterface *)
	interfaceQueryFailedAlarm :CNM_ConcreteMessages.TcError(event := Global.TC_EVENTS.MemoryErrors.MeasurementRecorderQueryInterfaceFailed , injectedService := THIS^.messageService);
	(* error for maximum queue size *)
	maxQueueSizeAlarm :CNM_ConcreteMessages.TcError(event := Global.TC_EVENTS.MemoryErrors.MeasurementsMaxQueueSize, injectedService := THIS^.messageService); 
END_VAR

(*
## Short summary

This methods creates a new measurement entry and queues it for the database insection.

.. <legal notes>

legal notes
=================
| SPDX-FileCopyrightText: © 2025 ekvip automation GmbH <info@ekvip.de>
| SPDX-License-Identifier: Apache-2.0
| For details check: Apache-2.0_

.. _Apache-2.0: https://www.apache.org/licenses/LICENSE-2.0

.. </legal notes>

*)
METHOD addMeasurementEntry :CNM_ReturnTypes.SingleExecutionResult;
VAR_INPUT
	(* product identifier for that specific part *)
	partIdentifier	:Tc2_System.T_MaxString;
	(* name of the measurement, e.g. label position, cell voltage, oven temperature *)
	name	: Tc2_System.T_MaxString;
	(* unit of the measurement, e.g. mm, V, °C *)
	unit	: CNM_ProductionMetricInterfaces.UnitString;
	(* Permissible value range of the measurement for OK parts*)
	range	: CNM_ProductionMetricInterfaces.MeasurementRangeStruct;
	(* value of the measurement *)
	value	: LREAL;
END_VAR
VAR
	dataset :CNM_ProductionMetricInterfaces.MeasurementEntryStruct;
	dto :POINTER TO MeasurementData := 0;
END_VAR
addMeasurementEntry := CNM_ReturnTypes.SingleExecutionResult.ABORTED;
// check if we can queue the dataset - throw error if the max queuesize is reached
IF ( THIS^.dataSetList.size >= THIS^.maxQueueSize ) THEN
	THIS^.maxQueueSizeAlarm.throw();
	RETURN;
END_IF

dataset.process := THIS^.configuration.process;
dataset.productType := THIS^.configuration.productType;
dataset.partIdentifier := partIdentifier;
dataset.name := name;
dataset.unit := unit;
dataset.range := range;
dataset.value := value;
dataset.timestamp := GetCurrentLTimeStamp();
dto := __NEW(MeasurementData(data := dataset));
IF (dto <> 0) THEN
	THIS^.dataSetList.append(dto^);
	addMeasurementEntry := CNM_ReturnTypes.SingleExecutionResult.SUCCESS;
END_IF
END_METHOD

(*

## Short summary

This abstract property returns the class name of the concrete object, 
which is useful for logging/debugging purpose or to check the class name
for ``__DELETE`` in factories (sometimes it's necessary to do more 
than just to free the memory).

.. <legal notes>

legal notes
=================
| SPDX-FileCopyrightText: © 2022 ekvip automation GmbH <info@ekvip.de>
| SPDX-License-Identifier: Apache-2.0
| For details check: Apache-2.0_

.. _Apache-2.0: https://www.apache.org/licenses/LICENSE-2.0

.. </legal notes>

*)
PROPERTY className : CNM_AbstractObject.ClassName
GET
className := 'MeasurementRecorder';
END_GET
END_PROPERTY

(* 
## Short summary

This is a fluent interface that provides single attempt commands, which can be evaluated by a cycle manager instance.
### Example 
```
	
	// execute command when leaving a step 
	cycleManager.leave(
		measurement.commands.addMeasurementEntry(
			partIdentifier	:= 'Part123',
			name := 'Voltage Check',
			unit := 'V',
			range := productType.VoltageCheck.Range,
			value := 3.14
		)
	); 
```	

.. <legal notes>

legal notes
=================
| SPDX-FileCopyrightText: © 2025 ekvip automation GmbH <info@ekvip.de>
| SPDX-License-Identifier: Apache-2.0
| For details check: Apache-2.0_

.. _Apache-2.0: https://www.apache.org/licenses/LICENSE-2.0

.. </legal notes>
	
*)
PROPERTY commands : CNM_ProductionMetricInterfaces.IMeasurementRecorderCommands
GET
commands := THIS^.measurementCommands;
END_GET
END_PROPERTY

(*
## Short summary

This property returns an fluent interface for the measurement configuration.
The following things should be configured after a type / product change was performed:
 -product type: either the name of the overall product or the individual feed parts to be processed
 
 
The process name can be set once during the initialization of the PLC as it usually doesn't change.

.. <legal notes>

legal notes
=================
| SPDX-FileCopyrightText: © 2022 ekvip automation GmbH <info@ekvip.de>
| SPDX-License-Identifier: Apache-2.0
| For details check: Apache-2.0_

.. _Apache-2.0: https://www.apache.org/licenses/LICENSE-2.0

.. </legal notes>

*)
PROPERTY configuration : CNM_ProductionMetricInterfaces.IProductionMetricsConfiguration
GET
VAR_INST
	config :DefaultMeasurementConfiguration;
END_VAR
configuration := config;
END_GET
END_PROPERTY

(* 
## Short summary

This method disables a node (E.g. axes should be disabled). It can take mutliple cycles. It has to be implemented for every node/device.
The execute input needs a rising edge to execute the method.
If there is nothing to disable, just return a 'SUCCESS' state.

This method is called automatically by the operation mode handler.

.. <legal notes>

legal notes
=================
| SPDX-FileCopyrightText: © 2024 ekvip automation GmbH <info@ekvip.de>
| SPDX-License-Identifier: Apache-2.0
| For details check: Apache-2.0_

.. _Apache-2.0: https://www.apache.org/licenses/LICENSE-2.0

.. </legal notes>

*)
METHOD disable : CNM_ReturnTypes.SingleExecutionState
VAR_INPUT
	execute	: BOOL;
END_VAR
// nothing to disable
disable := CNM_ReturnTypes.SingleExecutionState.SUCCESS;
END_METHOD

(* 
## Short summary

This method enables a node. It can take mutliple cycles. It has to be implemented for every node/device.
The intention is to enable devices here, e.g. axes, laser, dispenser etc.
The execute input needs a rising edge to execute the method.
If there is nothing to enable, just return a 'SUCCESS' state.

This method is called automatically by the operation mode handler.

.. <legal notes>

legal notes
=================
| SPDX-FileCopyrightText: © 2024 ekvip automation GmbH <info@ekvip.de>
| SPDX-License-Identifier: Apache-2.0
| For details check: Apache-2.0_

.. _Apache-2.0: https://www.apache.org/licenses/LICENSE-2.0

.. </legal notes>

*)
METHOD enable : CNM_ReturnTypes.SingleExecutionState
VAR_INPUT
	execute	: BOOL;
END_VAR
// nothing to enable
enable := CNM_ReturnTypes.SingleExecutionState.SUCCESS;
END_METHOD

(*

## Short summary

The constructor ``FB_init`` is needed to create an unique hash code.
The hash code is a pseudo random number create with a [xorshift](https://en.wikipedia.org/wiki/Xorshift) algorithm.
It can be overwritten on derivations, because it will be called implicit, ``SUPER^.FB_init()`` is not required.
For more information check: [Behavoir with derived function blocks](https://infosys.beckhoff.com/content/1033/tc3_plc_intro/5482088715.html?id=6983869892358031022)

.. <legal notes>

legal notes
=================
| SPDX-FileCopyrightText: © 2022 ekvip automation GmbH <info@ekvip.de>
| SPDX-License-Identifier: Apache-2.0
| For details check: Apache-2.0_

.. _Apache-2.0: https://www.apache.org/licenses/LICENSE-2.0

.. </legal notes>



*)
METHOD FB_init : BOOL
VAR_INPUT
	(* if TRUE, the retain variables are initialized (warm start / cold start)*)
	bInitRetains	: BOOL;
	(* if TRUE, the instance afterwards gets moved into the copy code (online change) *)
	bInCopyCode	:BOOL;
	(* the node were this node should be appended to *)
	parentNode :CNM_OpModeHandler.INodeInitialization;
END_VAR
THIS^.hmiInfo.template := 'MeasurementRecorder';
THIS^.isInHome := TRUE;
END_METHOD

(* 
## Short summary

This method contains instructions and sequences for the init mode. 
This mode is intended for initializing a machine, e.g. loading product type data from recipes, establish a connection to global production systems (MES).
If the node should do nothing, return a 'SUCCESS'.
It should run until all initializations are done or the mode is stopped immedtiately or a stop request is raised (THIS^.modeControl.stopRequest). 
This method is called automatically by the operation mode handler.

**Attention:** If this method returns the state 'ERROR', the operation mode handler automatically disables the whole machine! 

.. <legal notes>

legal notes
=================
| SPDX-FileCopyrightText: © 2024 ekvip automation GmbH <info@ekvip.de>
| SPDX-License-Identifier: Apache-2.0
| For details check: Apache-2.0_

.. _Apache-2.0: https://www.apache.org/licenses/LICENSE-2.0

.. </legal notes>

*)
METHOD initialize : CNM_ReturnTypes.SingleExecutionState
VAR_INPUT
	execute	: BOOL;
END_VAR
THIS^.measurementCommands.setRecorder(THIS^);
initialize := CNM_ReturnTypes.SingleExecutionState.SUCCESS;
END_METHOD

(*
## Short summary

This property getter returns the maximum queue size for the data recorder. 
If the dataset list has reached this size, no other dataset will be stored and an alarm will be raised.
For this class the maximum queue size can be configured as library parameter ''QUEUE_SIZE_FOR_DATA_RECORDS_PER_RECORDER''.
Overwrite this property for extended classes as the default implementation accesses the Parameter List of the CNM_ProductionMetrics library! 

.. <legal notes>

legal notes
=================
| SPDX-FileCopyrightText: © 2022 ekvip automation GmbH <info@ekvip.de>
| SPDX-License-Identifier: Apache-2.0
| For details check: Apache-2.0_

.. _Apache-2.0: https://www.apache.org/licenses/LICENSE-2.0

.. </legal notes>

*)

PROPERTY PROTECTED maxQueueSize : UDINT
GET
maxQueueSize := Settings.QUEUE_SIZE_FOR_DATA_RECORDS_PER_RECORDER;
END_GET
END_PROPERTY

(* 
## Short summary

This method will be called in every cycle for a node. It can be used to implement hardware drivers/measurements/monitoring.
The returned state defines the overall state of the node. It should return BUSY when the node executes a command, otherwise SUCCESS( or IDLE if there is nothing to do). 
(Simple monitoring is not a command an should return SUCCESS).  


**Attention:** the returned SingleExecutionState will be evaluated cyclically wihtin the node tree. 
In case a node returns an ERROR state, the whole machine will be disabled. 
Return ERROR only for fatal or critical errors and handle other errors within the node.
 

.. <legal notes>

legal notes
=================
| SPDX-FileCopyrightText: © 2025 ekvip automation GmbH <info@ekvip.de>
| SPDX-License-Identifier: Apache-2.0
| For details check: Apache-2.0_

.. _Apache-2.0: https://www.apache.org/licenses/LICENSE-2.0

.. </legal notes>
	
*)
METHOD run : CNM_ReturnTypes.SingleExecutionState
VAR_INST
	cycleManager :CNM_CycleManager.SimpleCycleManager;
END_VAR
VAR CONSTANT
	WAIT_FOR_DATA :DINT := 10;
	SET_DATA :DINT := 11;
	DATA_ERROR :DINT:= 12;
	WAIT_DATA_RECEIVED :DINT := 13;
END_VAR
VAR
	data :CNM_ProductionMetricInterfaces.IMeasurementData;
END_VAR
cycleManager(execute := TRUE);

CASE cycleManager.step.current OF
CNM_ReturnTypes.DefaultSteps.STEP.INIT:
	run := CNM_ReturnTypes.SingleExecutionState.SUCCESS;
	cycleManager.proceedWith(WAIT_FOR_DATA);
WAIT_FOR_DATA:
	run := CNM_ReturnTypes.SingleExecutionState.SUCCESS;
	IF (THIS^.dataSetList.size > 0) THEN
		run := CNM_ReturnTypes.SingleExecutionState.BUSY;
		cycleManager.proceedWith(SET_DATA); 
	END_IF
SET_DATA:
	run := CNM_ReturnTypes.SingleExecutionState.BUSY;
	IF (__QUERYINTERFACE(THIS^.dataSetList.dequeue(), data)) THEN
		(* fill dataslot *)
		THIS^.measurement := data.dataset;
		(* delete DTO *)
		data.destruct();
		(* set mailbox flag *)
		THIS^.newDataAvailable := TRUE;
		cycleManager.proceedWith(WAIT_DATA_RECEIVED);
	ELSE
		cycleManager.proceedWith(DATA_ERROR);
	END_IF
DATA_ERROR:
	cycleManager.step.next := SET_DATA;
	cycleManager.handle(THIS^.interfaceQueryFailedAlarm);
WAIT_DATA_RECEIVED:
	run := CNM_ReturnTypes.SingleExecutionState.BUSY;
	IF (NOT THIS^.newDataAvailable) THEN
		// clear data slot
		Tc2_System.MEMSET(destAddr := ADR(THIS^.measurement), 0, SIZEOF(THIS^.measurement));
		run := CNM_ReturnTypes.SingleExecutionState.SUCCESS;
		cycleManager.proceedWith(WAIT_FOR_DATA);
	END_IF
END_CASE
END_METHOD

(* 
## Short summary

This method executes stops all movements of a node. It has to be overwritten for every node. 
E.g. axes should perform a quickstop, cylinders should be turned off, etc.
If the node should do nothing, return a 'SUCCESS'.
It should stop axes/cylinders/process (e.g. laser welding, dispensing) endless until the manual mode is stopped via stop request or immediate stop.
This method is called automatically by the operation mode handler before disabling the machine or if the operator selects an immediate stop.

**Attention:** If this method returns the state 'ERROR', the operation mode handler automatically disables the whole machine! 

.. <legal notes>

legal notes
=================
| SPDX-FileCopyrightText: © 2024 ekvip automation GmbH <info@ekvip.de>
| SPDX-License-Identifier: Apache-2.0
| For details check: Apache-2.0_

.. _Apache-2.0: https://www.apache.org/licenses/LICENSE-2.0

.. </legal notes>

*)
METHOD stopImmediate : CNM_ReturnTypes.SingleExecutionState
VAR_INPUT
	execute	: BOOL;
END_VAR
// nothing to stop
stopImmediate := CNM_ReturnTypes.SingleExecutionState.SUCCESS;
END_METHOD

END_FUNCTION_BLOCK

// ---- Project Information/F_GetCompany.TcPOU
// This function has been automatically generated from the project information.
{attribute 'signature_flag' := '1073741824'}
{attribute 'TcGenerated'}
{attribute 'no-analysis'}
FUNCTION F_GetCompany : WSTRING
VAR_INPUT
	
END_VAR

F_GetCompany := "ekvip automation GmbH";

END_FUNCTION

// ---- Project Information/F_GetTitle.TcPOU
// This function has been automatically generated from the project information.
{attribute 'signature_flag' := '1073741824'}
{attribute 'TcGenerated'}
{attribute 'no-analysis'}
FUNCTION F_GetTitle : WSTRING
VAR_INPUT
	
END_VAR

F_GetTitle := "CNM Production Metrics";

END_FUNCTION

// ---- Project Information/F_GetVersion.TcPOU
// This function has been automatically generated from the project information.
{attribute 'signature_flag' := '1073741824'}
{attribute 'TcGenerated'}
{attribute 'no-analysis'}
FUNCTION F_GetVersion : ST_LibVersion
VAR_INPUT
	
END_VAR

F_GetVersion.iMajor := 1;
F_GetVersion.iMinor := 0;
F_GetVersion.iBuild := 0;
F_GetVersion.iRevision := 0;
F_GetVersion.sVersion := '1.0.0.0';
F_GetVersion.nFlags := 0;

END_FUNCTION
